LIN {X 0,Y 418.29,Z 497.008,A -85,B 0,C 180,E1 -10307.775,E2 -10307.775} C_VEL
LIN {X 0,Y 418.266,Z 497.012,A -85,B 0,C 180,E1 -10311.561,E2 -10311.561} C_VEL
LIN {X 0,Y 418.259,Z 497.011,A -85,B 0,C 180,E1 -10315.16,E2 -10315.16} C_VEL
LIN {X 0,Y 418.245,Z 497.014,A -85,B 0,C 180,E1 -10317.473,E2 -10317.473} C_VEL
LIN {X 0,Y 418.269,Z 497.007,A -85,B 0,C 180,E1 -10320.897,E2 -10320.897} C_VEL
LIN {X 0,Y 418.273,Z 497.008,A -85,B 0,C 180,E1 -10324.097,E2 -10324.097} C_VEL
LIN {X 0,Y 418.241,Z 497.014,A -85,B 0,C 180,E1 -10327.265,E2 -10327.265} C_VEL
LIN {X 0,Y 418.286,Z 497.005,A -85,B 0,C 180,E1 -10330.365,E2 -10330.365} C_VEL
LIN {X 0,Y 418.321,Z 497.004,A -85,B 0,C 180,E1 -10333.406,E2 -10333.406} C_VEL
LIN {X 0,Y 418.35,Z 496.998,A -85,B 0,C 180,E1 -10337,E2 -10337} C_VEL
LIN {X 0,Y 418.343,Z 496.998,A -85,B 0,C 180,E1 -10340.329,E2 -10340.329} C_VEL
LIN {X 0,Y 418.484,Z 496.982,A -85,B 0,C 180,E1 -10343.249,E2 -10343.249} C_VEL
LIN {X 0,Y 418.346,Z 496.999,A -85,B 0,C 180,E1 -10345.182,E2 -10345.182} C_VEL
LIN {X 0,Y 418.551,Z 496.974,A -85,B 0,C 180,E1 -10348.076,E2 -10348.076} C_VEL
LIN {X 0,Y 418.676,Z 496.959,A -85,B 0,C 180,E1 -10350,E2 -10350} C_VEL
LIN {X 0,Y 418.488,Z 496.984,A -85,B 0,C 180,E1 -10351.925,E2 -10351.925} C_VEL
LIN {X 0,Y 417.982,Z 497.048,A -85,B 0,C 180,E1 -10355.79,E2 -10355.79} C_VEL
LIN {X 0,Y 417.84,Z 497.118,A -85,B 0,C 180,E1 -10357.078,E2 -10357.078} C_VEL
LIN {X 0,Y 417.635,Z 500.157,A -85,B 0,C 180,E1 -10360.668,E2 -10360.668} C_VEL
LIN {X 0,Y 417.571,Z 502.391,A -85,B 0,C 180,E1 -10363.273,E2 -10363.273} C_VEL
LIN {X 0,Y 416.857,Z 502.803,A -85,B 0,C 180,E1 -10363.658,E2 -10363.658} C_VEL
LIN {X 0,Y 411.137,Z 504.383,A -85,B 0,C 180,E1 -10364.787,E2 -10364.787} C_VEL
LIN {X 0,Y 410.464,Z 504.792,A -85,B 0,C 180,E1 -10365.181,E2 -10365.181} C_VEL
LIN {X 0,Y 410.481,Z 505.038,A -85,B 0,C 180,E1 -10365.231,E2 -10365.231} C_VEL
LIN {X 0,Y 415.933,Z 520.618,A -85,B 0,C 180,E1 -10366,E2 -10366} C_VEL
LIN {X 0,Y 420.083,Z 534.2,A -85,B 0,C 180,E1 -10366.799,E2 -10366.799} C_VEL
LIN {X 0,Y 420.651,Z 537.197,A -85,B 0,C 180,E1 -10366.982,E2 -10366.982} C_VEL
LIN {X 0,Y 419.692,Z 552.291,A -85,B 0,C 180,E1 -10367.795,E2 -10367.795} C_VEL
LIN {X 0,Y 418.574,Z 565.955,A -85,B 0,C 180,E1 -10368.731,E2 -10368.731} C_VEL
LIN {X 0,Y 417.384,Z 578.751,A -85,B 0,C 180,E1 -10369.808,E2 -10369.808} C_VEL
LIN {X 0,Y 416.168,Z 591.539,A -85,B 0,C 180,E1 -10371.123,E2 -10371.123} C_VEL
LIN {X 0,Y 414.855,Z 603.015,A -85,B 0,C 180,E1 -10372.538,E2 -10372.538} C_VEL
LIN {X 0,Y 413.778,Z 613.302,A -85,B 0,C 180,E1 -10374.057,E2 -10374.057} C_VEL
LIN {X 0,Y 412.843,Z 621.821,A -85,B 0,C 180,E1 -10375.544,E2 -10375.544} C_VEL
LIN {X 0,Y 411.877,Z 630.973,A -85,B 0,C 180,E1 -10377.464,E2 -10377.464} C_VEL
LIN {X 0,Y 411.217,Z 638.263,A -85,B 0,C 180,E1 -10379.351,E2 -10379.351} C_VEL
LIN {X 0,Y 410.699,Z 643.934,A -85,B 0,C 180,E1 -10381.171,E2 -10381.171} C_VEL
LIN {X 0,Y 410.352,Z 648.94,A -85,B 0,C 180,E1 -10383.234,E2 -10383.234} C_VEL
LIN {X 0,Y 410.153,Z 651.623,A -85,B 0,C 180,E1 -10384.665,E2 -10384.665} C_VEL
LIN {X 0,Y 409.926,Z 654.472,A -85,B 0,C 180,E1 -10386.874,E2 -10386.874} C_VEL
LIN {X 0,Y 409.853,Z 655.422,A -85,B 0,C 180,E1 -10388.12,E2 -10388.12} C_VEL
LIN {X 0,Y 409.822,Z 655.948,A -85,B 0,C 180,E1 -10389.492,E2 -10389.492} C_VEL
LIN {X 0,Y 409.818,Z 655.929,A -85,B 0,C 180,E1 -10391.012,E2 -10391.012} C_VEL
LIN {X 0,Y 409.94,Z 654.61,A -85,B 0,C 180,E1 -10393.295,E2 -10393.295} C_VEL
LIN {X 0,Y 410.191,Z 652.038,A -85,B 0,C 180,E1 -10395.374,E2 -10395.374} C_VEL
LIN {X 0,Y 410.483,Z 648.227,A -85,B 0,C 180,E1 -10397.41,E2 -10397.41} C_VEL
LIN {X 0,Y 410.871,Z 643.027,A -85,B 0,C 180,E1 -10399.458,E2 -10399.458} C_VEL
LIN {X 0,Y 411.466,Z 636.994,A -85,B 0,C 180,E1 -10401.311,E2 -10401.311} C_VEL
LIN {X 0,Y 412.263,Z 629.191,A -85,B 0,C 180,E1 -10403.247,E2 -10403.247} C_VEL
LIN {X 0,Y 413.262,Z 620.342,A -85,B 0,C 180,E1 -10405.038,E2 -10405.038} C_VEL
LIN {X 0,Y 414.431,Z 610.328,A -85,B 0,C 180,E1 -10406.715,E2 -10406.715} C_VEL
LIN {X 0,Y 415.711,Z 599.27,A -85,B 0,C 180,E1 -10408.253,E2 -10408.253} C_VEL
LIN {X 0,Y 416.999,Z 587.412,A -85,B 0,C 180,E1 -10409.627,E2 -10409.627} C_VEL
LIN {X 0,Y 418.3,Z 574.278,A -85,B 0,C 180,E1 -10410.887,E2 -10410.887} C_VEL
LIN {X 0,Y 419.54,Z 560.488,A -85,B 0,C 180,E1 -10411.959,E2 -10411.959} C_VEL
LIN {X 0,Y 420.653,Z 546.6,A -85,B 0,C 180,E1 -10412.816,E2 -10412.816} C_VEL
LIN {X 0,Y 421.231,Z 537.263,A -85,B 0,C 180,E1 -10413.29,E2 -10413.29} C_VEL
LIN {X 0,Y 416.905,Z 523.396,A -85,B 0,C 180,E1 -10414.172,E2 -10414.172} C_VEL
LIN {X 0,Y 411.456,Z 509.384,A -85,B 0,C 180,E1 -10414.974,E2 -10414.974} C_VEL
LIN {X 0,Y 410.649,Z 506.752,A -85,B 0,C 180,E1 -10415.101,E2 -10415.101} C_VEL
LIN {X 0,Y 410.744,Z 504.603,A -85,B 0,C 180,E1 -10417.887,E2 -10417.887} C_VEL
LIN {X 0,Y 410.827,Z 502.253,A -85,B 0,C 180,E1 -10421.032,E2 -10421.032} C_VEL
LIN {X 0,Y 410.975,Z 499.978,A -85,B 0,C 180,E1 -10424.12,E2 -10424.12} C_VEL
LIN {X 0,Y 411.131,Z 497.904,A -85,B 0,C 180,E1 -10427.16,E2 -10427.16} C_VEL
LIN {X 0,Y 411.281,Z 497.883,A -85,B 0,C 180,E1 -10430.161,E2 -10430.161} C_VEL
LIN {X 0,Y 411.454,Z 497.857,A -85,B 0,C 180,E1 -10433.133,E2 -10433.133} C_VEL
LIN {X 0,Y 411.311,Z 497.876,A -85,B 0,C 180,E1 -10435.099,E2 -10435.099} C_VEL
LIN {X 0,Y 411.511,Z 497.851,A -85,B 0,C 180,E1 -10438.042,E2 -10438.042} C_VEL
LIN {X 0,Y 411.638,Z 497.835,A -85,B 0,C 180,E1 -10440,E2 -10440} C_VEL
LIN {X 0,Y 411.463,Z 497.858,A -85,B 0,C 180,E1 -10442.937,E2 -10442.937} C_VEL
LIN {X 0,Y 411.458,Z 497.859,A -85,B 0,C 180,E1 -10446.867,E2 -10446.867} C_VEL
LIN {X 0,Y 411.29,Z 497.877,A -85,B 0,C 180,E1 -10449.838,E2 -10449.838} C_VEL
LIN {X 0,Y 411.302,Z 497.876,A -85,B 0,C 180,E1 -10453.104,E2 -10453.104} C_VEL
LIN {X 0,Y 411.254,Z 497.882,A -85,B 0,C 180,E1 -10456.889,E2 -10456.889} C_VEL
LIN {X 0,Y 411.227,Z 497.884,A -85,B 0,C 180,E1 -10459.987,E2 -10459.987} C_VEL
LIN {X 0,Y 411.2,Z 497.887,A -85,B 0,C 180,E1 -10463.147,E2 -10463.147} C_VEL
LIN {X 0,Y 411.235,Z 497.885,A -85,B 0,C 180,E1 -10466.381,E2 -10466.381} C_VEL
LIN {X 0,Y 411.208,Z 497.891,A -85,B 0,C 180,E1 -10469.712,E2 -10469.712} C_VEL
LIN {X 0,Y 411.203,Z 497.889,A -85,B 0,C 180,E1 -10473.156,E2 -10473.156} C_VEL
LIN {X 0,Y 411.193,Z 497.892,A -85,B 0,C 180,E1 -10476.553,E2 -10476.553} C_VEL
LIN {X 0,Y 411.248,Z 498.032,A -85,B 0,C 180,E1 -10478.505,E2 -10478.505} C_VEL
LIN {X 0,Y 411.843,Z 501.621,A -85,B 0,C 180,E1 -10481.337,E2 -10481.337} C_VEL
LIN {X 0,Y 412.589,Z 505.831,A -85,B 0,C 180,E1 -10484.323,E2 -10484.323} C_VEL
LIN {X 0,Y 413.331,Z 510.237,A -85,B 0,C 180,E1 -10487.146,E2 -10487.146} C_VEL
LIN {X 0,Y 413.307,Z 513.645,A -85,B 0,C 180,E1 -10489.106,E2 -10489.106} C_VEL
LIN {X 0,Y 412.761,Z 519.39,A -85,B 0,C 180,E1 -10492.196,E2 -10492.196} C_VEL
LIN {X 0,Y 412.409,Z 524.702,A -85,B 0,C 180,E1 -10494.883,E2 -10494.883} C_VEL
LIN {X 0,Y 411.873,Z 532.35,A -85,B 0,C 180,E1 -10498.558,E2 -10498.558} C_VEL
LIN {X 0,Y 411.33,Z 539.833,A -85,B 0,C 180,E1 -10501.974,E2 -10501.974} C_VEL
LIN {X 0,Y 411.01,Z 546.461,A -85,B 0,C 180,E1 -10504.896,E2 -10504.896} C_VEL
LIN {X 0,Y 415.846,Z 565.472,A -85,B 0,C 180,E1 -10505.733,E2 -10505.733} C_VEL
LIN {X 0,Y 418.491,Z 580.052,A -85,B 0,C 180,E1 -10506.49,E2 -10506.49} C_VEL
LIN {X 0,Y 419.824,Z 589.116,A -85,B 0,C 180,E1 -10507.031,E2 -10507.031} C_VEL
LIN {X 0,Y 418.737,Z 602.749,A -85,B 0,C 180,E1 -10507.817,E2 -10507.817} C_VEL
LIN {X 0,Y 417.438,Z 616.129,A -85,B 0,C 180,E1 -10508.778,E2 -10508.778} C_VEL
LIN {X 0,Y 416.019,Z 629.933,A -85,B 0,C 180,E1 -10509.995,E2 -10509.995} C_VEL
LIN {X 0,Y 414.819,Z 641.407,A -85,B 0,C 180,E1 -10511.222,E2 -10511.222} C_VEL
LIN {X 0,Y 413.666,Z 653.061,A -85,B 0,C 180,E1 -10512.703,E2 -10512.703} C_VEL
LIN {X 0,Y 412.578,Z 662.893,A -85,B 0,C 180,E1 -10514.184,E2 -10514.184} C_VEL
LIN {X 0,Y 411.665,Z 672.58,A -85,B 0,C 180,E1 -10515.92,E2 -10515.92} C_VEL
LIN {X 0,Y 411.043,Z 680.676,A -85,B 0,C 180,E1 -10517.659,E2 -10517.659} C_VEL
LIN {X 0,Y 410.483,Z 688.249,A -85,B 0,C 180,E1 -10519.643,E2 -10519.643} C_VEL
LIN {X 0,Y 410.212,Z 694.284,A -85,B 0,C 180,E1 -10521.626,E2 -10521.626} C_VEL
LIN {X 0,Y 410.041,Z 699.25,A -85,B 0,C 180,E1 -10523.775,E2 -10523.775} C_VEL
LIN {X 0,Y 410.021,Z 701.523,A -85,B 0,C 180,E1 -10525.083,E2 -10525.083} C_VEL
LIN {X 0,Y 410.028,Z 703.932,A -85,B 0,C 180,E1 -10527.052,E2 -10527.052} C_VEL
LIN {X 0,Y 410.033,Z 705.156,A -85,B 0,C 180,E1 -10529.017,E2 -10529.017} C_VEL
LIN {X 0,Y 410.032,Z 705.191,A -85,B 0,C 180,E1 -10530.982,E2 -10530.982} C_VEL
LIN {X 0,Y 410.024,Z 704.011,A -85,B 0,C 180,E1 -10532.947,E2 -10532.947} C_VEL
LIN {X 0,Y 410.024,Z 701.648,A -85,B 0,C 180,E1 -10534.916,E2 -10534.916} C_VEL
LIN {X 0,Y 410.153,Z 698.06,A -85,B 0,C 180,E1 -10536.888,E2 -10536.888} C_VEL
LIN {X 0,Y 410.248,Z 693.142,A -85,B 0,C 180,E1 -10538.869,E2 -10538.869} C_VEL
LIN {X 0,Y 410.638,Z 686.783,A -85,B 0,C 180,E1 -10540.851,E2 -10540.851} C_VEL
LIN {X 0,Y 411.134,Z 678.795,A -85,B 0,C 180,E1 -10542.839,E2 -10542.839} C_VEL
LIN {X 0,Y 411.958,Z 670.307,A -85,B 0,C 180,E1 -10544.573,E2 -10544.573} C_VEL
LIN {X 0,Y 412.9,Z 660.081,A -85,B 0,C 180,E1 -10546.31,E2 -10546.31} C_VEL
LIN {X 0,Y 414.012,Z 649.665,A -85,B 0,C 180,E1 -10547.791,E2 -10547.791} C_VEL
LIN {X 0,Y 415.268,Z 637.192,A -85,B 0,C 180,E1 -10549.269,E2 -10549.269} C_VEL
LIN {X 0,Y 416.626,Z 624.734,A -85,B 0,C 180,E1 -10550.488,E2 -10550.488} C_VEL
LIN {X 0,Y 417.864,Z 611.122,A -85,B 0,C 180,E1 -10551.586,E2 -10551.586} C_VEL
LIN {X 0,Y 419.106,Z 597.196,A -85,B 0,C 180,E1 -10552.485,E2 -10552.485} C_VEL
LIN {X 0,Y 419.69,Z 588.951,A -85,B 0,C 180,E1 -10552.926,E2 -10552.926} C_VEL
LIN {X 0,Y 417.021,Z 573.601,A -85,B 0,C 180,E1 -10553.778,E2 -10553.778} C_VEL
LIN {X 0,Y 413.563,Z 558.078,A -85,B 0,C 180,E1 -10554.484,E2 -10554.484} C_VEL
LIN {X 0,Y 411.101,Z 548.197,A -85,B 0,C 180,E1 -10554.882,E2 -10554.882} C_VEL
LIN {X 0,Y 411.514,Z 541.099,A -85,B 0,C 180,E1 -10558.011,E2 -10558.011} C_VEL
LIN {X 0,Y 411.951,Z 533.541,A -85,B 0,C 180,E1 -10561.459,E2 -10561.459} C_VEL
LIN {X 0,Y 412.393,Z 527.674,A -85,B 0,C 180,E1 -10564.22,E2 -10564.22} C_VEL
LIN {X 0,Y 412.94,Z 520.375,A -85,B 0,C 180,E1 -10567.783,E2 -10567.783} C_VEL
LIN {X 0,Y 413.502,Z 514.296,A -85,B 0,C 180,E1 -10570.869,E2 -10570.869} C_VEL
LIN {X 0,Y 413.407,Z 510.324,A -85,B 0,C 180,E1 -10573.029,E2 -10573.029} C_VEL
LIN {X 0,Y 412.446,Z 504.612,A -85,B 0,C 180,E1 -10576.361,E2 -10576.361} C_VEL
LIN {X 0,Y 411.547,Z 499.514,A -85,B 0,C 180,E1 -10579.54,E2 -10579.54} C_VEL
LIN {X 0,Y 411.245,Z 497.886,A -85,B 0,C 180,E1 -10580.646,E2 -10580.646} C_VEL
LIN {X 0,Y 411.191,Z 497.891,A -85,B 0,C 180,E1 -10584.471,E2 -10584.471} C_VEL
LIN {X 0,Y 411.198,Z 497.89,A -85,B 0,C 180,E1 -10586.873,E2 -10586.873} C_VEL
LIN {X 0,Y 411.231,Z 497.883,A -85,B 0,C 180,E1 -10590.642,E2 -10590.642} C_VEL
LIN {X 0,Y 411.228,Z 497.888,A -85,B 0,C 180,E1 -10593.619,E2 -10593.619} C_VEL
LIN {X 0,Y 411.187,Z 497.89,A -85,B 0,C 180,E1 -10596.852,E2 -10596.852} C_VEL
LIN {X 0,Y 411.205,Z 497.888,A -85,B 0,C 180,E1 -10600.05,E2 -10600.05} C_VEL
LIN {X 0,Y 411.254,Z 497.883,A -85,B 0,C 180,E1 -10603.13,E2 -10603.13} C_VEL
LIN {X 0,Y 411.303,Z 497.875,A -85,B 0,C 180,E1 -10606.891,E2 -10606.891} C_VEL
LIN {X 0,Y 411.299,Z 497.876,A -85,B 0,C 180,E1 -10610.162,E2 -10610.162} C_VEL
LIN {X 0,Y 411.451,Z 497.859,A -85,B 0,C 180,E1 -10613.133,E2 -10613.133} C_VEL
LIN {X 0,Y 411.307,Z 497.876,A -85,B 0,C 180,E1 -10615.099,E2 -10615.099} C_VEL
LIN {X 0,Y 411.504,Z 497.851,A -85,B 0,C 180,E1 -10618.043,E2 -10618.043} C_VEL
LIN {X 0,Y 411.634,Z 497.835,A -85,B 0,C 180,E1 -10620,E2 -10620} C_VEL
LIN {X 0,Y 411.46,Z 497.856,A -85,B 0,C 180,E1 -10622.938,E2 -10622.938} C_VEL
LIN {X 0,Y 411.446,Z 497.856,A -85,B 0,C 180,E1 -10626.596,E2 -10626.596} C_VEL
LIN {X 0,Y 411.285,Z 497.88,A -85,B 0,C 180,E1 -10629.839,E2 -10629.839} C_VEL
LIN {X 0,Y 411.296,Z 497.878,A -85,B 0,C 180,E1 -10633.105,E2 -10633.105} C_VEL
LIN {X 0,Y 411.249,Z 497.881,A -85,B 0,C 180,E1 -10636.89,E2 -10636.89} C_VEL
LIN {X 0,Y 411.222,Z 497.887,A -85,B 0,C 180,E1 -10639.988,E2 -10639.988} C_VEL
LIN {X 0,Y 411.196,Z 497.891,A -85,B 0,C 180,E1 -10643.148,E2 -10643.148} C_VEL
LIN {X 0,Y 411.231,Z 497.883,A -85,B 0,C 180,E1 -10646.382,E2 -10646.382} C_VEL
LIN {X 0,Y 411.205,Z 497.891,A -85,B 0,C 180,E1 -10649.713,E2 -10649.713} C_VEL
LIN {X 0,Y 411.201,Z 497.89,A -85,B 0,C 180,E1 -10653.157,E2 -10653.157} C_VEL
LIN {X 0,Y 411.191,Z 497.888,A -85,B 0,C 180,E1 -10656.554,E2 -10656.554} C_VEL
LIN {X 0,Y 411.226,Z 497.889,A -85,B 0,C 180,E1 -10659.732,E2 -10659.732} C_VEL
LIN {X 0,Y 411.228,Z 497.886,A -85,B 0,C 180,E1 -10663.127,E2 -10663.127} C_VEL
LIN {X 0,Y 411.228,Z 497.887,A -85,B 0,C 180,E1 -10665.873,E2 -10665.873} C_VEL
LIN {X 0,Y 411.208,Z 497.886,A -85,B 0,C 180,E1 -10668.766,E2 -10668.766} C_VEL
LIN {X 0,Y 411.204,Z 497.889,A -85,B 0,C 180,E1 -10672.029,E2 -10672.029} C_VEL
LIN {X 0,Y 411.206,Z 497.891,A -85,B 0,C 180,E1 -10675.668,E2 -10675.668} C_VEL
LIN {X 0,Y 411.19,Z 497.891,A -85,B 0,C 180,E1 -10679.154,E2 -10679.154} C_VEL
LIN {X 0,Y 411.26,Z 497.88,A -85,B 0,C 180,E1 -10682.524,E2 -10682.524} C_VEL
LIN {X 0,Y 411.229,Z 497.888,A -85,B 0,C 180,E1 -10685.786,E2 -10685.786} C_VEL
LIN {X 0,Y 411.199,Z 497.888,A -85,B 0,C 180,E1 -10688.967,E2 -10688.967} C_VEL
LIN {X 0,Y 411.256,Z 497.882,A -85,B 0,C 180,E1 -10692.086,E2 -10692.086} C_VEL
LIN {X 0,Y 411.264,Z 497.881,A -85,B 0,C 180,E1 -10695.148,E2 -10695.148} C_VEL
LIN {X 0,Y 411.287,Z 497.878,A -85,B 0,C 180,E1 -10698.168,E2 -10698.168} C_VEL
LIN {X 0,Y 411.443,Z 497.858,A -85,B 0,C 180,E1 -10702.192,E2 -10702.192} C_VEL
LIN {X 0,Y 411.476,Z 497.855,A -85,B 0,C 180,E1 -10704.119,E2 -10704.119} C_VEL
LIN {X 0,Y 411.52,Z 497.85,A -85,B 0,C 180,E1 -10708.043,E2 -10708.043} C_VEL
LIN {X 0,Y 411.645,Z 497.835,A -85,B 0,C 180,E1 -10710,E2 -10710} C_VEL
LIN {X 0,Y 411.45,Z 497.86,A -85,B 0,C 180,E1 -10711.958,E2 -10711.958} C_VEL
LIN {X 0,Y 410.941,Z 497.924,A -85,B 0,C 180,E1 -10715.89,E2 -10715.89} C_VEL
LIN {X 0,Y 410.799,Z 497.969,A -85,B 0,C 180,E1 -10717.123,E2 -10717.123} C_VEL
LIN {X 0,Y 410.621,Z 500.232,A -85,B 0,C 180,E1 -10719.855,E2 -10719.855} C_VEL
LIN {X 0,Y 410.538,Z 502.812,A -85,B 0,C 180,E1 -10722.859,E2 -10722.859} C_VEL
LIN {X 0,Y 410.464,Z 504.792,A -85,B 0,C 180,E1 -10725.181,E2 -10725.181} C_VEL
LIN {X 0,Y 411.369,Z 505.402,A -85,B 0,C 180,E1 -10725.295,E2 -10725.295} C_VEL
LIN {X 0,Y 414.064,Z 508.494,A -85,B 0,C 180,E1 -10725.536,E2 -10725.536} C_VEL
LIN {X 0,Y 415.611,Z 511.968,A -85,B 0,C 180,E1 -10725.706,E2 -10725.706} C_VEL
LIN {X 0,Y 416.194,Z 517.03,A -85,B 0,C 180,E1 -10725.897,E2 -10725.897} C_VEL
LIN {X 0,Y 415.635,Z 521.611,A -85,B 0,C 180,E1 -10725.95,E2 -10725.95} C_VEL
LIN {X 0,Y 413.296,Z 529.526,A -85,B 0,C 180,E1 -10726.151,E2 -10726.151} C_VEL
LIN {X 0,Y 412.906,Z 532.831,A -85,B 0,C 180,E1 -10726.3,E2 -10726.3} C_VEL
LIN {X 0,Y 413.193,Z 534.941,A -85,B 0,C 180,E1 -10726.425,E2 -10726.425} C_VEL
LIN {X 0,Y 414.006,Z 538.808,A -85,B 0,C 180,E1 -10726.673,E2 -10726.673} C_VEL
LIN {X 0,Y 413.055,Z 553.102,A -85,B 0,C 180,E1 -10727.466,E2 -10727.466} C_VEL
LIN {X 0,Y 411.911,Z 566.481,A -85,B 0,C 180,E1 -10728.4,E2 -10728.4} C_VEL
LIN {X 0,Y 410.608,Z 579.831,A -85,B 0,C 180,E1 -10729.55,E2 -10729.55} C_VEL
LIN {X 0,Y 409.376,Z 592.351,A -85,B 0,C 180,E1 -10730.869,E2 -10730.869} C_VEL
LIN {X 0,Y 408.042,Z 603.489,A -85,B 0,C 180,E1 -10732.267,E2 -10732.267} C_VEL
LIN {X 0,Y 406.935,Z 613.382,A -85,B 0,C 180,E1 -10733.744,E2 -10733.744} C_VEL
LIN {X 0,Y 405.887,Z 622.569,A -85,B 0,C 180,E1 -10735.376,E2 -10735.376} C_VEL
LIN {X 0,Y 404.946,Z 631.301,A -85,B 0,C 180,E1 -10737.245,E2 -10737.245} C_VEL
LIN {X 0,Y 404.221,Z 638.5,A -85,B 0,C 180,E1 -10739.132,E2 -10739.132} C_VEL
LIN {X 0,Y 403.705,Z 643.887,A -85,B 0,C 180,E1 -10740.869,E2 -10740.869} C_VEL
LIN {X 0,Y 403.351,Z 648.436,A -85,B 0,C 180,E1 -10742.693,E2 -10742.693} C_VEL
LIN {X 0,Y 403.191,Z 650.843,A -85,B 0,C 180,E1 -10743.903,E2 -10743.903} C_VEL
LIN {X 0,Y 403.006,Z 652.842,A -85,B 0,C 180,E1 -10745.133,E2 -10745.133} C_VEL
LIN {X 0,Y 402.849,Z 654.698,A -85,B 0,C 180,E1 -10746.629,E2 -10746.629} C_VEL
LIN {X 0,Y 402.757,Z 656.254,A -85,B 0,C 180,E1 -10748.916,E2 -10748.916} C_VEL
LIN {X 0,Y 402.724,Z 656.466,A -85,B 0,C 180,E1 -10750.217,E2 -10750.217} C_VEL
LIN {X 0,Y 402.745,Z 656.187,A -85,B 0,C 180,E1 -10751.537,E2 -10751.537} C_VEL
LIN {X 0,Y 402.838,Z 655.408,A -85,B 0,C 180,E1 -10752.883,E2 -10752.883} C_VEL
LIN {X 0,Y 402.976,Z 653.999,A -85,B 0,C 180,E1 -10754.352,E2 -10754.352} C_VEL
LIN {X 0,Y 403.263,Z 650.841,A -85,B 0,C 180,E1 -10756.454,E2 -10756.454} C_VEL
LIN {X 0,Y 403.651,Z 646.288,A -85,B 0,C 180,E1 -10758.576,E2 -10758.576} C_VEL
LIN {X 0,Y 404.185,Z 640.494,A -85,B 0,C 180,E1 -10760.617,E2 -10760.617} C_VEL
LIN {X 0,Y 404.943,Z 633.389,A -85,B 0,C 180,E1 -10762.594,E2 -10762.594} C_VEL
LIN {X 0,Y 405.921,Z 625.107,A -85,B 0,C 180,E1 -10764.463,E2 -10764.463} C_VEL
LIN {X 0,Y 407.058,Z 615.553,A -85,B 0,C 180,E1 -10766.241,E2 -10766.241} C_VEL
LIN {X 0,Y 408.388,Z 604.754,A -85,B 0,C 180,E1 -10767.904,E2 -10767.904} C_VEL
LIN {X 0,Y 409.742,Z 593.312,A -85,B 0,C 180,E1 -10769.367,E2 -10769.367} C_VEL
LIN {X 0,Y 411.097,Z 580.984,A -85,B 0,C 180,E1 -10770.677,E2 -10770.677} C_VEL
LIN {X 0,Y 412.434,Z 567.966,A -85,B 0,C 180,E1 -10771.814,E2 -10771.814} C_VEL
LIN {X 0,Y 413.63,Z 554.227,A -85,B 0,C 180,E1 -10772.787,E2 -10772.787} C_VEL
LIN {X 0,Y 414.649,Z 539.89,A -85,B 0,C 180,E1 -10773.586,E2 -10773.586} C_VEL
LIN {X 0,Y 414.021,Z 536.459,A -85,B 0,C 180,E1 -10773.809,E2 -10773.809} C_VEL
LIN {X 0,Y 409.117,Z 521.383,A -85,B 0,C 180,E1 -10774.791,E2 -10774.791} C_VEL
LIN {X 0,Y 403.693,Z 507.937,A -85,B 0,C 180,E1 -10775.576,E2 -10775.576} C_VEL
LIN {X 0,Y 403.588,Z 507.237,A -85,B 0,C 180,E1 -10775.638,E2 -10775.638} C_VEL
LIN {X 0,Y 403.718,Z 505.038,A -85,B 0,C 180,E1 -10778.557,E2 -10778.557} C_VEL
LIN {X 0,Y 403.838,Z 502.696,A -85,B 0,C 180,E1 -10781.744,E2 -10781.744} C_VEL
LIN {X 0,Y 403.983,Z 500.441,A -85,B 0,C 180,E1 -10784.873,E2 -10784.873} C_VEL
LIN {X 0,Y 404.078,Z 499.029,A -85,B 0,C 180,E1 -10786.932,E2 -10786.932} C_VEL
LIN {X 0,Y 404.208,Z 498.764,A -85,B 0,C 180,E1 -10788.973,E2 -10788.973} C_VEL
LIN {X 0,Y 404.403,Z 498.738,A -85,B 0,C 180,E1 -10792.128,E2 -10792.128} C_VEL
LIN {X 0,Y 404.421,Z 498.736,A -85,B 0,C 180,E1 -10794.015,E2 -10794.015} C_VEL
LIN {X 0,Y 404.48,Z 498.727,A -85,B 0,C 180,E1 -10798.008,E2 -10798.008} C_VEL
LIN {X 0,Y 404.608,Z 498.711,A -85,B 0,C 180,E1 -10800,E2 -10800} C_VEL
LIN {X 0,Y 404.42,Z 498.735,A -85,B 0,C 180,E1 -10802.988,E2 -10802.988} C_VEL
LIN {X 0,Y 404.409,Z 498.736,A -85,B 0,C 180,E1 -10806.987,E2 -10806.987} C_VEL
LIN {X 0,Y 404.256,Z 498.753,A -85,B 0,C 180,E1 -10810.011,E2 -10810.011} C_VEL
LIN {X 0,Y 404.263,Z 498.752,A -85,B 0,C 180,E1 -10813.211,E2 -10813.211} C_VEL
LIN {X 0,Y 404.212,Z 498.758,A -85,B 0,C 180,E1 -10817.007,E2 -10817.007} C_VEL
LIN {X 0,Y 404.16,Z 498.768,A -85,B 0,C 180,E1 -10820.351,E2 -10820.351} C_VEL
LIN {X 0,Y 404.166,Z 498.763,A -85,B 0,C 180,E1 -10823.574,E2 -10823.574} C_VEL
LIN {X 0,Y 404.181,Z 498.764,A -85,B 0,C 180,E1 -10825.766,E2 -10825.766} C_VEL
LIN {X 0,Y 404.195,Z 498.764,A -85,B 0,C 180,E1 -10827.999,E2 -10827.999} C_VEL
LIN {X 0,Y 404.14,Z 498.77,A -85,B 0,C 180,E1 -10831.559,E2 -10831.559} C_VEL
LIN {X 0,Y 404.183,Z 498.764,A -85,B 0,C 180,E1 -10835.016,E2 -10835.016} C_VEL
LIN {X 0,Y 404.167,Z 498.875,A -85,B 0,C 180,E1 -10837.888,E2 -10837.888} C_VEL
LIN {X 0,Y 404.69,Z 501.567,A -85,B 0,C 180,E1 -10840.172,E2 -10840.172} C_VEL
LIN {X 0,Y 405.524,Z 506.611,A -85,B 0,C 180,E1 -10843.886,E2 -10843.886} C_VEL
LIN {X 0,Y 406.233,Z 510.723,A -85,B 0,C 180,E1 -10846.603,E2 -10846.603} C_VEL
LIN {X 0,Y 406.408,Z 513.041,A -85,B 0,C 180,E1 -10848.038,E2 -10848.038} C_VEL
LIN {X 0,Y 405.925,Z 518.639,A -85,B 0,C 180,E1 -10851.179,E2 -10851.179} C_VEL
LIN {X 0,Y 405.422,Z 525.101,A -85,B 0,C 180,E1 -10854.562,E2 -10854.562} C_VEL
LIN {X 0,Y 404.945,Z 530.94,A -85,B 0,C 180,E1 -10857.451,E2 -10857.451} C_VEL
LIN {X 0,Y 404.548,Z 536.955,A -85,B 0,C 180,E1 -10860.299,E2 -10860.299} C_VEL
LIN {X 0,Y 404.099,Z 544.343,A -85,B 0,C 180,E1 -10863.673,E2 -10863.673} C_VEL
LIN {X 0,Y 403.992,Z 545.989,A -85,B 0,C 180,E1 -10864.408,E2 -10864.408} C_VEL
LIN {X 0,Y 408.505,Z 563.256,A -85,B 0,C 180,E1 -10865.187,E2 -10865.187} C_VEL
LIN {X 0,Y 411.418,Z 577.948,A -85,B 0,C 180,E1 -10865.967,E2 -10865.967} C_VEL
LIN {X 0,Y 413.168,Z 590.212,A -85,B 0,C 180,E1 -10866.713,E2 -10866.713} C_VEL
LIN {X 0,Y 411.923,Z 604.633,A -85,B 0,C 180,E1 -10867.586,E2 -10867.586} C_VEL
LIN {X 0,Y 410.628,Z 617.372,A -85,B 0,C 180,E1 -10868.541,E2 -10868.541} C_VEL
LIN {X 0,Y 409.15,Z 630.825,A -85,B 0,C 180,E1 -10869.776,E2 -10869.776} C_VEL
LIN {X 0,Y 407.829,Z 642.875,A -85,B 0,C 180,E1 -10871.113,E2 -10871.113} C_VEL
LIN {X 0,Y 406.606,Z 654.458,A -85,B 0,C 180,E1 -10872.653,E2 -10872.653} C_VEL
LIN {X 0,Y 405.371,Z 665.473,A -85,B 0,C 180,E1 -10874.411,E2 -10874.411} C_VEL
LIN {X 0,Y 404.471,Z 674.794,A -85,B 0,C 180,E1 -10876.203,E2 -10876.203} C_VEL
LIN {X 0,Y 403.838,Z 682.334,A -85,B 0,C 180,E1 -10877.946,E2 -10877.946} C_VEL
LIN {X 0,Y 403.286,Z 689.494,A -85,B 0,C 180,E1 -10879.964,E2 -10879.964} C_VEL
LIN {X 0,Y 403.078,Z 695.147,A -85,B 0,C 180,E1 -10881.981,E2 -10881.981} C_VEL
LIN {X 0,Y 402.936,Z 699.433,A -85,B 0,C 180,E1 -10883.992,E2 -10883.992} C_VEL
LIN {X 0,Y 402.879,Z 702.449,A -85,B 0,C 180,E1 -10885.998,E2 -10885.998} C_VEL
LIN {X 0,Y 402.971,Z 704.265,A -85,B 0,C 180,E1 -10888.001,E2 -10888.001} C_VEL
LIN {X 0,Y 402.963,Z 704.904,A -85,B 0,C 180,E1 -10889.999,E2 -10889.999} C_VEL
LIN {X 0,Y 402.97,Z 704.32,A -85,B 0,C 180,E1 -10891.998,E2 -10891.998} C_VEL
LIN {X 0,Y 402.87,Z 702.543,A -85,B 0,C 180,E1 -10894.001,E2 -10894.001} C_VEL
LIN {X 0,Y 402.984,Z 699.573,A -85,B 0,C 180,E1 -10896.006,E2 -10896.006} C_VEL
LIN {X 0,Y 403.078,Z 695.324,A -85,B 0,C 180,E1 -10898.017,E2 -10898.017} C_VEL
LIN {X 0,Y 403.286,Z 689.692,A -85,B 0,C 180,E1 -10900.035,E2 -10900.035} C_VEL
LIN {X 0,Y 403.839,Z 682.539,A -85,B 0,C 180,E1 -10902.053,E2 -10902.053} C_VEL
LIN {X 0,Y 404.475,Z 675.009,A -85,B 0,C 180,E1 -10903.796,E2 -10903.796} C_VEL
LIN {X 0,Y 405.373,Z 665.673,A -85,B 0,C 180,E1 -10905.588,E2 -10905.588} C_VEL
LIN {X 0,Y 406.639,Z 654.56,A -85,B 0,C 180,E1 -10907.345,E2 -10907.345} C_VEL
LIN {X 0,Y 407.825,Z 642.842,A -85,B 0,C 180,E1 -10908.888,E2 -10908.888} C_VEL
LIN {X 0,Y 409.14,Z 630.638,A -85,B 0,C 180,E1 -10910.223,E2 -10910.223} C_VEL
LIN {X 0,Y 410.411,Z 618.372,A -85,B 0,C 180,E1 -10911.338,E2 -10911.338} C_VEL
LIN {X 0,Y 411.844,Z 603.969,A -85,B 0,C 180,E1 -10912.402,E2 -10912.402} C_VEL
LIN {X 0,Y 412.988,Z 589.857,A -85,B 0,C 180,E1 -10913.229,E2 -10913.229} C_VEL
LIN {X 0,Y 410.247,Z 573.892,A -85,B 0,C 180,E1 -10914.149,E2 -10914.149} C_VEL
LIN {X 0,Y 406.646,Z 557.983,A -85,B 0,C 180,E1 -10914.9,E2 -10914.9} C_VEL
LIN {X 0,Y 404.09,Z 547.804,A -85,B 0,C 180,E1 -10915.312,E2 -10915.312} C_VEL
LIN {X 0,Y 404.502,Z 540.697,A -85,B 0,C 180,E1 -10918.54,E2 -10918.54} C_VEL
LIN {X 0,Y 404.93,Z 533.843,A -85,B 0,C 180,E1 -10921.74,E2 -10921.74} C_VEL
LIN {X 0,Y 405.365,Z 528.511,A -85,B 0,C 180,E1 -10924.295,E2 -10924.295} C_VEL
LIN {X 0,Y 406.084,Z 520.002,A -85,B 0,C 180,E1 -10928.537,E2 -10928.537} C_VEL
LIN {X 0,Y 406.513,Z 515.155,A -85,B 0,C 180,E1 -10931.067,E2 -10931.067} C_VEL
LIN {X 0,Y 406.336,Z 510.917,A -85,B 0,C 180,E1 -10933.412,E2 -10933.412} C_VEL
LIN {X 0,Y 405.354,Z 505.371,A -85,B 0,C 180,E1 -10936.733,E2 -10936.733} C_VEL
LIN {X 0,Y 404.457,Z 500.266,A -85,B 0,C 180,E1 -10939.99,E2 -10939.99} C_VEL
LIN {X 0,Y 404.174,Z 498.767,A -85,B 0,C 180,E1 -10941.086,E2 -10941.086} C_VEL
LIN {X 0,Y 404.177,Z 498.764,A -85,B 0,C 180,E1 -10944.983,E2 -10944.983} C_VEL
LIN {X 0,Y 404.137,Z 498.767,A -85,B 0,C 180,E1 -10948.554,E2 -10948.554} C_VEL
LIN {X 0,Y 404.189,Z 498.762,A -85,B 0,C 180,E1 -10952,E2 -10952} C_VEL
LIN {X 0,Y 404.165,Z 498.768,A -85,B 0,C 180,E1 -10955.334,E2 -10955.334} C_VEL
LIN {X 0,Y 404.128,Z 498.768,A -85,B 0,C 180,E1 -10958.58,E2 -10958.58} C_VEL
LIN {X 0,Y 404.2,Z 498.763,A -85,B 0,C 180,E1 -10961.762,E2 -10961.762} C_VEL
LIN {X 0,Y 404.202,Z 498.759,A -85,B 0,C 180,E1 -10964.882,E2 -10964.882} C_VEL
LIN {X 0,Y 404.26,Z 498.754,A -85,B 0,C 180,E1 -10967.959,E2 -10967.959} C_VEL
LIN {X 0,Y 404.423,Z 498.732,A -85,B 0,C 180,E1 -10972.1,E2 -10972.1} C_VEL
LIN {X 0,Y 404.416,Z 498.733,A -85,B 0,C 180,E1 -10974.015,E2 -10974.015} C_VEL
LIN {X 0,Y 404.473,Z 498.727,A -85,B 0,C 180,E1 -10978.009,E2 -10978.009} C_VEL
LIN {X 0,Y 404.603,Z 498.711,A -85,B 0,C 180,E1 -10980,E2 -10980} C_VEL
LIN {X 0,Y 404.417,Z 498.733,A -85,B 0,C 180,E1 -10982.989,E2 -10982.989} C_VEL
LIN {X 0,Y 404.394,Z 498.734,A -85,B 0,C 180,E1 -10986.593,E2 -10986.593} C_VEL
LIN {X 0,Y 404.282,Z 498.75,A -85,B 0,C 180,E1 -10989.002,E2 -10989.002} C_VEL
LIN {X 0,Y 404.248,Z 498.755,A -85,B 0,C 180,E1 -10992.042,E2 -10992.042} C_VEL
LIN {X 0,Y 404.197,Z 498.762,A -85,B 0,C 180,E1 -10995.119,E2 -10995.119} C_VEL
LIN {X 0,Y 404.202,Z 498.759,A -85,B 0,C 180,E1 -10998.239,E2 -10998.239} C_VEL
LIN {X 0,Y 404.131,Z 498.772,A -85,B 0,C 180,E1 -11001.42,E2 -11001.42} C_VEL
LIN {X 0,Y 404.17,Z 498.763,A -85,B 0,C 180,E1 -11004.667,E2 -11004.667} C_VEL
LIN {X 0,Y 404.191,Z 498.762,A -85,B 0,C 180,E1 -11008.001,E2 -11008.001} C_VEL
LIN {X 0,Y 404.141,Z 498.772,A -85,B 0,C 180,E1 -11011.561,E2 -11011.561} C_VEL
LIN {X 0,Y 404.18,Z 498.763,A -85,B 0,C 180,E1 -11015.017,E2 -11015.017} C_VEL
LIN {X 0,Y 404.16,Z 498.764,A -85,B 0,C 180,E1 -11018.757,E2 -11018.757} C_VEL
LIN {X 0,Y 404.188,Z 498.765,A -85,B 0,C 180,E1 -11021.612,E2 -11021.612} C_VEL
LIN {X 0,Y 404.198,Z 498.759,A -85,B 0,C 180,E1 -11024.531,E2 -11024.531} C_VEL
LIN {X 0,Y 404.205,Z 498.762,A -85,B 0,C 180,E1 -11027.306,E2 -11027.306} C_VEL
LIN {X 0,Y 404.167,Z 498.766,A -85,B 0,C 180,E1 -11029.957,E2 -11029.957} C_VEL
LIN {X 0,Y 404.14,Z 498.769,A -85,B 0,C 180,E1 -11033.125,E2 -11033.125} C_VEL
LIN {X 0,Y 404.145,Z 498.767,A -85,B 0,C 180,E1 -11036.189,E2 -11036.189} C_VEL
LIN {X 0,Y 404.146,Z 498.771,A -85,B 0,C 180,E1 -11039.716,E2 -11039.716} C_VEL
LIN {X 0,Y 404.197,Z 498.761,A -85,B 0,C 180,E1 -11043.124,E2 -11043.124} C_VEL
LIN {X 0,Y 404.179,Z 498.765,A -85,B 0,C 180,E1 -11045.336,E2 -11045.336} C_VEL
LIN {X 0,Y 404.141,Z 498.766,A -85,B 0,C 180,E1 -11048.582,E2 -11048.582} C_VEL
LIN {X 0,Y 404.214,Z 498.762,A -85,B 0,C 180,E1 -11051.763,E2 -11051.763} C_VEL
LIN {X 0,Y 404.21,Z 498.758,A -85,B 0,C 180,E1 -11054.883,E2 -11054.883} C_VEL
LIN {X 0,Y 404.26,Z 498.755,A -85,B 0,C 180,E1 -11057.959,E2 -11057.959} C_VEL
LIN {X 0,Y 404.27,Z 498.751,A -85,B 0,C 180,E1 -11060.999,E2 -11060.999} C_VEL
LIN {X 0,Y 404.423,Z 498.734,A -85,B 0,C 180,E1 -11064.016,E2 -11064.016} C_VEL
LIN {X 0,Y 404.489,Z 498.726,A -85,B 0,C 180,E1 -11068.009,E2 -11068.009} C_VEL
LIN {X 0,Y 404.614,Z 498.71,A -85,B 0,C 180,E1 -11070.001,E2 -11070.001} C_VEL
LIN {X 0,Y 404.412,Z 498.736,A -85,B 0,C 180,E1 -11071.992,E2 -11071.992} C_VEL
LIN {X 0,Y 403.901,Z 498.801,A -85,B 0,C 180,E1 -11075.993,E2 -11075.993} C_VEL
LIN {X 0,Y 403.761,Z 498.823,A -85,B 0,C 180,E1 -11077.174,E2 -11077.174} C_VEL
LIN {X 0,Y 403.556,Z 501.208,A -85,B 0,C 180,E1 -11080.03,E2 -11080.03} C_VEL
LIN {X 0,Y 403.461,Z 503.783,A -85,B 0,C 180,E1 -11083.088,E2 -11083.088} C_VEL
LIN {X 0,Y 403.406,Z 505.213,A -85,B 0,C 180,E1 -11084.761,E2 -11084.761} C_VEL
LIN {X 0,Y 405.428,Z 511.037,A -85,B 0,C 180,E1 -11085.056,E2 -11085.056} C_VEL
LIN {X 0,Y 410.426,Z 525.605,A -85,B 0,C 180,E1 -11085.849,E2 -11085.849} C_VEL
LIN {X 0,Y 413.193,Z 534.941,A -85,B 0,C 180,E1 -11086.425,E2 -11086.425} C_VEL
LIN {X 0,Y 413.294,Z 537.952,A -85,B 0,C 180,E1 -11086.583,E2 -11086.583} C_VEL
LIN {X 0,Y 411.822,Z 542.242,A -85,B 0,C 180,E1 -11086.72,E2 -11086.72} C_VEL
LIN {X 0,Y 407.314,Z 550.681,A -85,B 0,C 180,E1 -11086.959,E2 -11086.959} C_VEL
LIN {X 0,Y 406.419,Z 554.435,A -85,B 0,C 180,E1 -11087.161,E2 -11087.161} C_VEL
LIN {X 0,Y 405.3,Z 566.721,A -85,B 0,C 180,E1 -11088.036,E2 -11088.036} C_VEL
LIN {X 0,Y 403.993,Z 579.74,A -85,B 0,C 180,E1 -11089.169,E2 -11089.169} C_VEL
LIN {X 0,Y 402.76,Z 591.653,A -85,B 0,C 180,E1 -11090.426,E2 -11090.426} C_VEL
LIN {X 0,Y 401.241,Z 603.807,A -85,B 0,C 180,E1 -11091.964,E2 -11091.964} C_VEL
LIN {X 0,Y 400.027,Z 614.253,A -85,B 0,C 180,E1 -11093.559,E2 -11093.559} C_VEL
LIN {X 0,Y 398.914,Z 623.458,A -85,B 0,C 180,E1 -11095.232,E2 -11095.232} C_VEL
LIN {X 0,Y 397.973,Z 631.754,A -85,B 0,C 180,E1 -11097.048,E2 -11097.048} C_VEL
LIN {X 0,Y 397.171,Z 639.466,A -85,B 0,C 180,E1 -11099.118,E2 -11099.118} C_VEL
LIN {X 0,Y 396.643,Z 644.846,A -85,B 0,C 180,E1 -11100.92,E2 -11100.92} C_VEL
LIN {X 0,Y 396.293,Z 649.193,A -85,B 0,C 180,E1 -11102.745,E2 -11102.745} C_VEL
LIN {X 0,Y 395.992,Z 652.609,A -85,B 0,C 180,E1 -11104.606,E2 -11104.606} C_VEL
LIN {X 0,Y 395.737,Z 655.445,A -85,B 0,C 180,E1 -11106.949,E2 -11106.949} C_VEL
LIN {X 0,Y 395.669,Z 656.526,A -85,B 0,C 180,E1 -11108.597,E2 -11108.597} C_VEL
LIN {X 0,Y 395.664,Z 656.897,A -85,B 0,C 180,E1 -11110.2,E2 -11110.2} C_VEL
LIN {X 0,Y 395.714,Z 656.217,A -85,B 0,C 180,E1 -11112.445,E2 -11112.445} C_VEL
LIN {X 0,Y 395.936,Z 654.052,A -85,B 0,C 180,E1 -11114.763,E2 -11114.763} C_VEL
LIN {X 0,Y 396.226,Z 651.158,A -85,B 0,C 180,E1 -11116.654,E2 -11116.654} C_VEL
LIN {X 0,Y 396.598,Z 647.111,A -85,B 0,C 180,E1 -11118.579,E2 -11118.579} C_VEL
LIN {X 0,Y 397.069,Z 642.167,A -85,B 0,C 180,E1 -11120.417,E2 -11120.417} C_VEL
LIN {X 0,Y 397.779,Z 636.056,A -85,B 0,C 180,E1 -11122.253,E2 -11122.253} C_VEL
LIN {X 0,Y 398.709,Z 628.186,A -85,B 0,C 180,E1 -11124.177,E2 -11124.177} C_VEL
LIN {X 0,Y 399.929,Z 618.612,A -85,B 0,C 180,E1 -11126.085,E2 -11126.085} C_VEL
LIN {X 0,Y 401.322,Z 607.996,A -85,B 0,C 180,E1 -11127.826,E2 -11127.826} C_VEL
LIN {X 0,Y 402.608,Z 597.656,A -85,B 0,C 180,E1 -11129.249,E2 -11129.249} C_VEL
LIN {X 0,Y 404.008,Z 586.014,A -85,B 0,C 180,E1 -11130.587,E2 -11130.587} C_VEL
LIN {X 0,Y 405.538,Z 572.164,A -85,B 0,C 180,E1 -11131.897,E2 -11131.897} C_VEL
LIN {X 0,Y 406.861,Z 558.154,A -85,B 0,C 180,E1 -11132.966,E2 -11132.966} C_VEL
LIN {X 0,Y 407.989,Z 544.296,A -85,B 0,C 180,E1 -11133.804,E2 -11133.804} C_VEL
LIN {X 0,Y 408.166,Z 541.316,A -85,B 0,C 180,E1 -11133.954,E2 -11133.954} C_VEL
LIN {X 0,Y 406.077,Z 533.341,A -85,B 0,C 180,E1 -11134.511,E2 -11134.511} C_VEL
LIN {X 0,Y 401.6,Z 520.387,A -85,B 0,C 180,E1 -11135.372,E2 -11135.372} C_VEL
LIN {X 0,Y 396.715,Z 508.613,A -85,B 0,C 180,E1 -11136.093,E2 -11136.093} C_VEL
LIN {X 0,Y 396.571,Z 507.764,A -85,B 0,C 180,E1 -11136.153,E2 -11136.153} C_VEL
LIN {X 0,Y 396.727,Z 505.023,A -85,B 0,C 180,E1 -11139.865,E2 -11139.865} C_VEL
LIN {X 0,Y 396.893,Z 502.403,A -85,B 0,C 180,E1 -11143.541,E2 -11143.541} C_VEL
LIN {X 0,Y 397.067,Z 500.169,A -85,B 0,C 180,E1 -11146.775,E2 -11146.775} C_VEL
LIN {X 0,Y 397.068,Z 499.656,A -85,B 0,C 180,E1 -11147.737,E2 -11147.737} C_VEL
LIN {X 0,Y 397.247,Z 499.628,A -85,B 0,C 180,E1 -11150.838,E2 -11150.838} C_VEL
LIN {X 0,Y 397.372,Z 499.614,A -85,B 0,C 180,E1 -11153.908,E2 -11153.908} C_VEL
LIN {X 0,Y 397.449,Z 499.603,A -85,B 0,C 180,E1 -11157.973,E2 -11157.973} C_VEL
LIN {X 0,Y 397.577,Z 499.587,A -85,B 0,C 180,E1 -11160,E2 -11160} C_VEL
LIN {X 0,Y 397.378,Z 499.612,A -85,B 0,C 180,E1 -11163.041,E2 -11163.041} C_VEL
LIN {X 0,Y 397.361,Z 499.613,A -85,B 0,C 180,E1 -11167.111,E2 -11167.111} C_VEL
LIN {X 0,Y 397.215,Z 499.63,A -85,B 0,C 180,E1 -11170.191,E2 -11170.191} C_VEL
LIN {X 0,Y 397.223,Z 499.628,A -85,B 0,C 180,E1 -11173.321,E2 -11173.321} C_VEL
LIN {X 0,Y 397.179,Z 499.634,A -85,B 0,C 180,E1 -11177.155,E2 -11177.155} C_VEL
LIN {X 0,Y 397.099,Z 499.646,A -85,B 0,C 180,E1 -11180.73,E2 -11180.73} C_VEL
LIN {X 0,Y 397.13,Z 499.643,A -85,B 0,C 180,E1 -11184.018,E2 -11184.018} C_VEL
LIN {X 0,Y 397.192,Z 499.634,A -85,B 0,C 180,E1 -11187.39,E2 -11187.39} C_VEL
LIN {X 0,Y 397.082,Z 499.65,A -85,B 0,C 180,E1 -11190.882,E2 -11190.882} C_VEL
LIN {X 0,Y 397.123,Z 499.643,A -85,B 0,C 180,E1 -11194.493,E2 -11194.493} C_VEL
LIN {X 0,Y 397.118,Z 499.673,A -85,B 0,C 180,E1 -11197.214,E2 -11197.214} C_VEL
LIN {X 0,Y 397.829,Z 503.577,A -85,B 0,C 180,E1 -11200.569,E2 -11200.569} C_VEL
LIN {X 0,Y 398.521,Z 507.746,A -85,B 0,C 180,E1 -11203.694,E2 -11203.694} C_VEL
LIN {X 0,Y 399.277,Z 512.106,A -85,B 0,C 180,E1 -11206.649,E2 -11206.649} C_VEL
LIN {X 0,Y 399.423,Z 514.351,A -85,B 0,C 180,E1 -11208.039,E2 -11208.039} C_VEL
LIN {X 0,Y 398.968,Z 519.18,A -85,B 0,C 180,E1 -11210.812,E2 -11210.812} C_VEL
LIN {X 0,Y 398.425,Z 525.869,A -85,B 0,C 180,E1 -11214.402,E2 -11214.402} C_VEL
LIN {X 0,Y 397.908,Z 531.808,A -85,B 0,C 180,E1 -11217.405,E2 -11217.405} C_VEL
LIN {X 0,Y 397.492,Z 537.831,A -85,B 0,C 180,E1 -11220.326,E2 -11220.326} C_VEL
LIN {X 0,Y 397.02,Z 545.439,A -85,B 0,C 180,E1 -11223.87,E2 -11223.87} C_VEL
LIN {X 0,Y 402.092,Z 564.819,A -85,B 0,C 180,E1 -11224.804,E2 -11224.804} C_VEL
LIN {X 0,Y 404.96,Z 579.748,A -85,B 0,C 180,E1 -11225.641,E2 -11225.641} C_VEL
LIN {X 0,Y 406.522,Z 591.325,A -85,B 0,C 180,E1 -11226.386,E2 -11226.386} C_VEL
LIN {X 0,Y 405.146,Z 606.244,A -85,B 0,C 180,E1 -11227.331,E2 -11227.331} C_VEL
LIN {X 0,Y 403.684,Z 619.951,A -85,B 0,C 180,E1 -11228.421,E2 -11228.421} C_VEL
LIN {X 0,Y 402.186,Z 632.879,A -85,B 0,C 180,E1 -11229.677,E2 -11229.677} C_VEL
LIN {X 0,Y 400.809,Z 644.706,A -85,B 0,C 180,E1 -11231.061,E2 -11231.061} C_VEL
LIN {X 0,Y 399.546,Z 655.746,A -85,B 0,C 180,E1 -11232.6,E2 -11232.6} C_VEL
LIN {X 0,Y 398.454,Z 665.074,A -85,B 0,C 180,E1 -11234.134,E2 -11234.134} C_VEL
LIN {X 0,Y 397.498,Z 674.265,A -85,B 0,C 180,E1 -11235.93,E2 -11235.93} C_VEL
LIN {X 0,Y 396.832,Z 681.924,A -85,B 0,C 180,E1 -11237.729,E2 -11237.729} C_VEL
LIN {X 0,Y 396.23,Z 689.081,A -85,B 0,C 180,E1 -11239.783,E2 -11239.783} C_VEL
LIN {X 0,Y 396.011,Z 694.733,A -85,B 0,C 180,E1 -11241.837,E2 -11241.837} C_VEL
LIN {X 0,Y 395.859,Z 699.015,A -85,B 0,C 180,E1 -11243.885,E2 -11243.885} C_VEL
LIN {X 0,Y 395.798,Z 702.028,A -85,B 0,C 180,E1 -11245.927,E2 -11245.927} C_VEL
LIN {X 0,Y 395.9,Z 703.841,A -85,B 0,C 180,E1 -11247.965,E2 -11247.965} C_VEL
LIN {X 0,Y 395.884,Z 704.476,A -85,B 0,C 180,E1 -11249.999,E2 -11249.999} C_VEL
LIN {X 0,Y 395.899,Z 703.891,A -85,B 0,C 180,E1 -11252.034,E2 -11252.034} C_VEL
LIN {X 0,Y 395.791,Z 702.106,A -85,B 0,C 180,E1 -11254.072,E2 -11254.072} C_VEL
LIN {X 0,Y 395.929,Z 698.863,A -85,B 0,C 180,E1 -11256.263,E2 -11256.263} C_VEL
LIN {X 0,Y 396.012,Z 694.866,A -85,B 0,C 180,E1 -11258.161,E2 -11258.161} C_VEL
LIN {X 0,Y 396.23,Z 689.217,A -85,B 0,C 180,E1 -11260.216,E2 -11260.216} C_VEL
LIN {X 0,Y 396.829,Z 682.045,A -85,B 0,C 180,E1 -11262.27,E2 -11262.27} C_VEL
LIN {X 0,Y 397.499,Z 674.372,A -85,B 0,C 180,E1 -11264.069,E2 -11264.069} C_VEL
LIN {X 0,Y 398.434,Z 665.142,A -85,B 0,C 180,E1 -11265.866,E2 -11265.866} C_VEL
LIN {X 0,Y 399.576,Z 655.728,A -85,B 0,C 180,E1 -11267.397,E2 -11267.397} C_VEL
LIN {X 0,Y 400.81,Z 644.504,A -85,B 0,C 180,E1 -11268.941,E2 -11268.941} C_VEL
LIN {X 0,Y 402.14,Z 632.459,A -85,B 0,C 180,E1 -11270.324,E2 -11270.324} C_VEL
LIN {X 0,Y 403.579,Z 619.171,A -85,B 0,C 180,E1 -11271.584,E2 -11271.584} C_VEL
LIN {X 0,Y 405.039,Z 605.177,A -85,B 0,C 180,E1 -11272.656,E2 -11272.656} C_VEL
LIN {X 0,Y 406.264,Z 590.862,A -85,B 0,C 180,E1 -11273.531,E2 -11273.531} C_VEL
LIN {X 0,Y 403.649,Z 575.364,A -85,B 0,C 180,E1 -11274.465,E2 -11274.465} C_VEL
LIN {X 0,Y 400.263,Z 560.095,A -85,B 0,C 180,E1 -11275.226,E2 -11275.226} C_VEL
LIN {X 0,Y 397.088,Z 547.442,A -85,B 0,C 180,E1 -11275.766,E2 -11275.766} C_VEL
LIN {X 0,Y 397.486,Z 540.259,A -85,B 0,C 180,E1 -11279.092,E2 -11279.092} C_VEL
LIN {X 0,Y 397.922,Z 534.093,A -85,B 0,C 180,E1 -11282.031,E2 -11282.031} C_VEL
LIN {X 0,Y 398.331,Z 529.33,A -85,B 0,C 180,E1 -11284.373,E2 -11284.373} C_VEL
LIN {X 0,Y 398.957,Z 522.036,A -85,B 0,C 180,E1 -11288.064,E2 -11288.064} C_VEL
LIN {X 0,Y 399.538,Z 515.872,A -85,B 0,C 180,E1 -11291.336,E2 -11291.336} C_VEL
LIN {X 0,Y 399.377,Z 512.335,A -85,B 0,C 180,E1 -11293.336,E2 -11293.336} C_VEL
LIN {X 0,Y 398.461,Z 507.057,A -85,B 0,C 180,E1 -11296.538,E2 -11296.538} C_VEL
LIN {X 0,Y 397.642,Z 502.503,A -85,B 0,C 180,E1 -11299.461,E2 -11299.461} C_VEL
LIN {X 0,Y 397.131,Z 499.643,A -85,B 0,C 180,E1 -11301.425,E2 -11301.425} C_VEL
LIN {X 0,Y 397.112,Z 499.644,A -85,B 0,C 180,E1 -11304.496,E2 -11304.496} C_VEL
LIN {X 0,Y 397.072,Z 499.649,A -85,B 0,C 180,E1 -11307.928,E2 -11307.928} C_VEL
LIN {X 0,Y 397.118,Z 499.646,A -85,B 0,C 180,E1 -11311.456,E2 -11311.456} C_VEL
LIN {X 0,Y 397.143,Z 499.638,A -85,B 0,C 180,E1 -11314.487,E2 -11314.487} C_VEL
LIN {X 0,Y 397.086,Z 499.646,A -85,B 0,C 180,E1 -11318.181,E2 -11318.181} C_VEL
LIN {X 0,Y 397.152,Z 499.642,A -85,B 0,C 180,E1 -11321.426,E2 -11321.426} C_VEL
LIN {X 0,Y 397.174,Z 499.634,A -85,B 0,C 180,E1 -11324.608,E2 -11324.608} C_VEL
LIN {X 0,Y 397.219,Z 499.633,A -85,B 0,C 180,E1 -11327.742,E2 -11327.742} C_VEL
LIN {X 0,Y 397.385,Z 499.609,A -85,B 0,C 180,E1 -11332.041,E2 -11332.041} C_VEL
LIN {X 0,Y 397.25,Z 499.625,A -85,B 0,C 180,E1 -11334.925,E2 -11334.925} C_VEL
LIN {X 0,Y 397.442,Z 499.603,A -85,B 0,C 180,E1 -11337.974,E2 -11337.974} C_VEL
LIN {X 0,Y 397.573,Z 499.586,A -85,B 0,C 180,E1 -11340,E2 -11340} C_VEL
LIN {X 0,Y 397.376,Z 499.611,A -85,B 0,C 180,E1 -11343.042,E2 -11343.042} C_VEL
LIN {X 0,Y 397.346,Z 499.612,A -85,B 0,C 180,E1 -11346.588,E2 -11346.588} C_VEL
LIN {X 0,Y 397.244,Z 499.628,A -85,B 0,C 180,E1 -11349.162,E2 -11349.162} C_VEL
LIN {X 0,Y 397.211,Z 499.63,A -85,B 0,C 180,E1 -11352.259,E2 -11352.259} C_VEL
LIN {X 0,Y 397.17,Z 499.639,A -85,B 0,C 180,E1 -11355.393,E2 -11355.393} C_VEL
LIN {X 0,Y 397.154,Z 499.636,A -85,B 0,C 180,E1 -11358.574,E2 -11358.574} C_VEL
LIN {X 0,Y 397.089,Z 499.649,A -85,B 0,C 180,E1 -11361.819,E2 -11361.819} C_VEL
LIN {X 0,Y 397.149,Z 499.639,A -85,B 0,C 180,E1 -11365.133,E2 -11365.133} C_VEL
LIN {X 0,Y 397.157,Z 499.64,A -85,B 0,C 180,E1 -11367.778,E2 -11367.778} C_VEL
LIN {X 0,Y 397.081,Z 499.646,A -85,B 0,C 180,E1 -11370.883,E2 -11370.883} C_VEL
LIN {X 0,Y 397.12,Z 499.641,A -85,B 0,C 180,E1 -11374.494,E2 -11374.494} C_VEL
LIN {X 0,Y 397.106,Z 499.643,A -85,B 0,C 180,E1 -11378.275,E2 -11378.275} C_VEL
LIN {X 0,Y 397.153,Z 499.639,A -85,B 0,C 180,E1 -11381.995,E2 -11381.995} C_VEL
LIN {X 0,Y 397.147,Z 499.639,A -85,B 0,C 180,E1 -11385.061,E2 -11385.061} C_VEL
LIN {X 0,Y 397.153,Z 499.639,A -85,B 0,C 180,E1 -11388.008,E2 -11388.008} C_VEL
LIN {X 0,Y 397.109,Z 499.647,A -85,B 0,C 180,E1 -11391.727,E2 -11391.727} C_VEL
LIN {X 0,Y 397.125,Z 499.645,A -85,B 0,C 180,E1 -11395.508,E2 -11395.508} C_VEL
LIN {X 0,Y 397.079,Z 499.648,A -85,B 0,C 180,E1 -11399.119,E2 -11399.119} C_VEL
LIN {X 0,Y 397.196,Z 499.631,A -85,B 0,C 180,E1 -11402.611,E2 -11402.611} C_VEL
LIN {X 0,Y 397.135,Z 499.642,A -85,B 0,C 180,E1 -11405.983,E2 -11405.983} C_VEL
LIN {X 0,Y 397.141,Z 499.643,A -85,B 0,C 180,E1 -11409.706,E2 -11409.706} C_VEL
LIN {X 0,Y 397.185,Z 499.633,A -85,B 0,C 180,E1 -11412.846,E2 -11412.846} C_VEL
LIN {X 0,Y 397.232,Z 499.627,A -85,B 0,C 180,E1 -11416.704,E2 -11416.704} C_VEL
LIN {X 0,Y 397.221,Z 499.632,A -85,B 0,C 180,E1 -11419.81,E2 -11419.81} C_VEL
LIN {X 0,Y 397.343,Z 499.613,A -85,B 0,C 180,E1 -11422.888,E2 -11422.888} C_VEL
LIN {X 0,Y 397.26,Z 499.624,A -85,B 0,C 180,E1 -11424.926,E2 -11424.926} C_VEL
LIN {X 0,Y 397.458,Z 499.602,A -85,B 0,C 180,E1 -11427.974,E2 -11427.974} C_VEL
LIN {X 0,Y 397.583,Z 499.586,A -85,B 0,C 180,E1 -11430.001,E2 -11430.001} C_VEL
LIN {X 0,Y 397.372,Z 499.612,A -85,B 0,C 180,E1 -11432.028,E2 -11432.028} C_VEL
LIN {X 0,Y 396.842,Z 499.679,A -85,B 0,C 180,E1 -11436.1,E2 -11436.1} C_VEL
LIN {X 0,Y 396.724,Z 499.703,A -85,B 0,C 180,E1 -11437.227,E2 -11437.227} C_VEL
LIN {X 0,Y 396.504,Z 502.158,A -85,B 0,C 180,E1 -11440.21,E2 -11440.21} C_VEL
LIN {X 0,Y 396.386,Z 504.767,A -85,B 0,C 180,E1 -11443.326,E2 -11443.326} C_VEL
LIN {X 0,Y 396.391,Z 505.821,A -85,B 0,C 180,E1 -11444.34,E2 -11444.34} C_VEL
LIN {X 0,Y 399.282,Z 513.904,A -85,B 0,C 180,E1 -11444.738,E2 -11444.738} C_VEL
LIN {X 0,Y 404.165,Z 528.288,A -85,B 0,C 180,E1 -11445.564,E2 -11445.564} C_VEL
LIN {X 0,Y 407.372,Z 539.664,A -85,B 0,C 180,E1 -11446.313,E2 -11446.313} C_VEL
LIN {X 0,Y 406.419,Z 554.435,A -85,B 0,C 180,E1 -11447.161,E2 -11447.161} C_VEL
LIN {X 0,Y 405.43,Z 559.796,A -85,B 0,C 180,E1 -11447.487,E2 -11447.487} C_VEL
LIN {X 0,Y 401.92,Z 568.4,A -85,B 0,C 180,E1 -11447.978,E2 -11447.978} C_VEL
LIN {X 0,Y 398.293,Z 576.786,A -85,B 0,C 180,E1 -11448.543,E2 -11448.543} C_VEL
LIN {X 0,Y 397.137,Z 581.678,A -85,B 0,C 180,E1 -11448.98,E2 -11448.98} C_VEL
LIN {X 0,Y 395.85,Z 593.744,A -85,B 0,C 180,E1 -11450.308,E2 -11450.308} C_VEL
LIN {X 0,Y 394.427,Z 604.441,A -85,B 0,C 180,E1 -11451.699,E2 -11451.699} C_VEL
LIN {X 0,Y 393.064,Z 615.516,A -85,B 0,C 180,E1 -11453.435,E2 -11453.435} C_VEL
LIN {X 0,Y 391.883,Z 624.919,A -85,B 0,C 180,E1 -11455.21,E2 -11455.21} C_VEL
LIN {X 0,Y 390.934,Z 632.809,A -85,B 0,C 180,E1 -11456.996,E2 -11456.996} C_VEL
LIN {X 0,Y 390.304,Z 638.596,A -85,B 0,C 180,E1 -11458.565,E2 -11458.565} C_VEL
LIN {X 0,Y 389.738,Z 644.035,A -85,B 0,C 180,E1 -11460.326,E2 -11460.326} C_VEL
LIN {X 0,Y 389.339,Z 648.186,A -85,B 0,C 180,E1 -11461.961,E2 -11461.961} C_VEL
LIN {X 0,Y 388.978,Z 652.284,A -85,B 0,C 180,E1 -11464.063,E2 -11464.063} C_VEL
LIN {X 0,Y 388.781,Z 654.473,A -85,B 0,C 180,E1 -11465.563,E2 -11465.563} C_VEL
LIN {X 0,Y 388.621,Z 656.639,A -85,B 0,C 180,E1 -11467.942,E2 -11467.942} C_VEL
LIN {X 0,Y 388.569,Z 657.188,A -85,B 0,C 180,E1 -11469.275,E2 -11469.275} C_VEL
LIN {X 0,Y 388.574,Z 657.276,A -85,B 0,C 180,E1 -11470.626,E2 -11470.626} C_VEL
LIN {X 0,Y 388.617,Z 656.827,A -85,B 0,C 180,E1 -11472.142,E2 -11472.142} C_VEL
LIN {X 0,Y 388.717,Z 655.76,A -85,B 0,C 180,E1 -11473.68,E2 -11473.68} C_VEL
LIN {X 0,Y 388.912,Z 654.049,A -85,B 0,C 180,E1 -11475.189,E2 -11475.189} C_VEL
LIN {X 0,Y 389.253,Z 650.762,A -85,B 0,C 180,E1 -11477.242,E2 -11477.242} C_VEL
LIN {X 0,Y 389.663,Z 646.397,A -85,B 0,C 180,E1 -11479.245,E2 -11479.245} C_VEL
LIN {X 0,Y 390.342,Z 640.667,A -85,B 0,C 180,E1 -11481.268,E2 -11481.268} C_VEL
LIN {X 0,Y 391.23,Z 633.355,A -85,B 0,C 180,E1 -11483.326,E2 -11483.326} C_VEL
LIN {X 0,Y 392.392,Z 624.743,A -85,B 0,C 180,E1 -11485.286,E2 -11485.286} C_VEL
LIN {X 0,Y 393.636,Z 615.357,A -85,B 0,C 180,E1 -11487.049,E2 -11487.049} C_VEL
LIN {X 0,Y 395.132,Z 604.397,A -85,B 0,C 180,E1 -11488.756,E2 -11488.756} C_VEL
LIN {X 0,Y 396.647,Z 592.787,A -85,B 0,C 180,E1 -11490.256,E2 -11490.256} C_VEL
LIN {X 0,Y 398.216,Z 579.793,A -85,B 0,C 180,E1 -11491.645,E2 -11491.645} C_VEL
LIN {X 0,Y 399.76,Z 565.227,A -85,B 0,C 180,E1 -11492.902,E2 -11492.902} C_VEL
LIN {X 0,Y 401.072,Z 551.72,A -85,B 0,C 180,E1 -11493.83,E2 -11493.83} C_VEL
LIN {X 0,Y 401.591,Z 541.895,A -85,B 0,C 180,E1 -11494.394,E2 -11494.394} C_VEL
LIN {X 0,Y 397.307,Z 528,A -85,B 0,C 180,E1 -11495.402,E2 -11495.402} C_VEL
LIN {X 0,Y 392.066,Z 514.637,A -85,B 0,C 180,E1 -11496.304,E2 -11496.304} C_VEL
LIN {X 0,Y 389.68,Z 509.049,A -85,B 0,C 180,E1 -11496.65,E2 -11496.65} C_VEL
LIN {X 0,Y 389.569,Z 508.269,A -85,B 0,C 180,E1 -11496.724,E2 -11496.724} C_VEL
LIN {X 0,Y 389.718,Z 505.925,A -85,B 0,C 180,E1 -11499.962,E2 -11499.962} C_VEL
LIN {X 0,Y 389.859,Z 503.63,A -85,B 0,C 180,E1 -11503.235,E2 -11503.235} C_VEL
LIN {X 0,Y 390.022,Z 501.295,A -85,B 0,C 180,E1 -11506.666,E2 -11506.666} C_VEL
LIN {X 0,Y 390.026,Z 500.754,A -85,B 0,C 180,E1 -11507.512,E2 -11507.512} C_VEL
LIN {X 0,Y 390.197,Z 500.507,A -85,B 0,C 180,E1 -11510.671,E2 -11510.671} C_VEL
LIN {X 0,Y 390.325,Z 500.492,A -85,B 0,C 180,E1 -11513.798,E2 -11513.798} C_VEL
LIN {X 0,Y 390.418,Z 500.479,A -85,B 0,C 180,E1 -11517.936,E2 -11517.936} C_VEL
LIN {X 0,Y 390.547,Z 500.462,A -85,B 0,C 180,E1 -11520,E2 -11520} C_VEL
LIN {X 0,Y 390.312,Z 500.492,A -85,B 0,C 180,E1 -11523.096,E2 -11523.096} C_VEL
LIN {X 0,Y 390.328,Z 500.489,A -85,B 0,C 180,E1 -11526.202,E2 -11526.202} C_VEL
LIN {X 0,Y 390.312,Z 500.491,A -85,B 0,C 180,E1 -11528.282,E2 -11528.282} C_VEL
LIN {X 0,Y 390.168,Z 500.51,A -85,B 0,C 180,E1 -11532.483,E2 -11532.483} C_VEL
LIN {X 0,Y 390.135,Z 500.511,A -85,B 0,C 180,E1 -11535.677,E2 -11535.677} C_VEL
LIN {X 0,Y 390.102,Z 500.516,A -85,B 0,C 180,E1 -11538.922,E2 -11538.922} C_VEL
LIN {X 0,Y 390.037,Z 500.527,A -85,B 0,C 180,E1 -11542.234,E2 -11542.234} C_VEL
LIN {X 0,Y 390.116,Z 500.516,A -85,B 0,C 180,E1 -11545.743,E2 -11545.743} C_VEL
LIN {X 0,Y 390.062,Z 500.523,A -85,B 0,C 180,E1 -11549.109,E2 -11549.109} C_VEL
LIN {X 0,Y 390.041,Z 500.526,A -85,B 0,C 180,E1 -11552.721,E2 -11552.721} C_VEL
LIN {X 0,Y 390.054,Z 500.524,A -85,B 0,C 180,E1 -11555.825,E2 -11555.825} C_VEL
LIN {X 0,Y 390.084,Z 500.76,A -85,B 0,C 180,E1 -11556.762,E2 -11556.762} C_VEL
LIN {X 0,Y 390.636,Z 503.58,A -85,B 0,C 180,E1 -11559.32,E2 -11559.32} C_VEL
LIN {X 0,Y 391.313,Z 507.659,A -85,B 0,C 180,E1 -11562.578,E2 -11562.578} C_VEL
LIN {X 0,Y 392.1,Z 512.189,A -85,B 0,C 180,E1 -11565.804,E2 -11565.804} C_VEL
LIN {X 0,Y 392.45,Z 515.371,A -85,B 0,C 180,E1 -11567.884,E2 -11567.884} C_VEL
LIN {X 0,Y 391.897,Z 520.946,A -85,B 0,C 180,E1 -11571.122,E2 -11571.122} C_VEL
LIN {X 0,Y 391.474,Z 525.957,A -85,B 0,C 180,E1 -11573.888,E2 -11573.888} C_VEL
LIN {X 0,Y 390.935,Z 531.45,A -85,B 0,C 180,E1 -11576.749,E2 -11576.749} C_VEL
LIN {X 0,Y 390.507,Z 537.475,A -85,B 0,C 180,E1 -11579.752,E2 -11579.752} C_VEL
LIN {X 0,Y 390.018,Z 544.964,A -85,B 0,C 180,E1 -11583.337,E2 -11583.337} C_VEL
LIN {X 0,Y 390.8,Z 548.09,A -85,B 0,C 180,E1 -11583.472,E2 -11583.472} C_VEL
LIN {X 0,Y 395.148,Z 564.237,A -85,B 0,C 180,E1 -11584.292,E2 -11584.292} C_VEL
LIN {X 0,Y 398.064,Z 578.716,A -85,B 0,C 180,E1 -11585.133,E2 -11585.133} C_VEL
LIN {X 0,Y 399.905,Z 592.448,A -85,B 0,C 180,E1 -11586.043,E2 -11586.043} C_VEL
LIN {X 0,Y 398.4,Z 607.696,A -85,B 0,C 180,E1 -11587.053,E2 -11587.053} C_VEL
LIN {X 0,Y 396.897,Z 621.108,A -85,B 0,C 180,E1 -11588.17,E2 -11588.17} C_VEL
LIN {X 0,Y 395.323,Z 633.749,A -85,B 0,C 180,E1 -11589.444,E2 -11589.444} C_VEL
LIN {X 0,Y 393.897,Z 645.54,A -85,B 0,C 180,E1 -11590.875,E2 -11590.875} C_VEL
LIN {X 0,Y 392.488,Z 657.046,A -85,B 0,C 180,E1 -11592.546,E2 -11592.546} C_VEL
LIN {X 0,Y 391.369,Z 666.087,A -85,B 0,C 180,E1 -11594.106,E2 -11594.106} C_VEL
LIN {X 0,Y 390.416,Z 675.025,A -85,B 0,C 180,E1 -11595.935,E2 -11595.935} C_VEL
LIN {X 0,Y 389.807,Z 681.523,A -85,B 0,C 180,E1 -11597.505,E2 -11597.505} C_VEL
LIN {X 0,Y 389.178,Z 688.668,A -85,B 0,C 180,E1 -11599.596,E2 -11599.596} C_VEL
LIN {X 0,Y 388.935,Z 694.319,A -85,B 0,C 180,E1 -11601.688,E2 -11601.688} C_VEL
LIN {X 0,Y 388.775,Z 698.74,A -85,B 0,C 180,E1 -11603.851,E2 -11603.851} C_VEL
LIN {X 0,Y 388.72,Z 701.607,A -85,B 0,C 180,E1 -11605.852,E2 -11605.852} C_VEL
LIN {X 0,Y 388.83,Z 703.417,A -85,B 0,C 180,E1 -11607.928,E2 -11607.928} C_VEL
LIN {X 0,Y 388.808,Z 704.047,A -85,B 0,C 180,E1 -11609.999,E2 -11609.999} C_VEL
LIN {X 0,Y 388.829,Z 703.46,A -85,B 0,C 180,E1 -11612.071,E2 -11612.071} C_VEL
LIN {X 0,Y 388.714,Z 701.665,A -85,B 0,C 180,E1 -11614.147,E2 -11614.147} C_VEL
LIN {X 0,Y 388.831,Z 698.675,A -85,B 0,C 180,E1 -11616.225,E2 -11616.225} C_VEL
LIN {X 0,Y 388.938,Z 694.401,A -85,B 0,C 180,E1 -11618.311,E2 -11618.311} C_VEL
LIN {X 0,Y 389.178,Z 688.737,A -85,B 0,C 180,E1 -11620.403,E2 -11620.403} C_VEL
LIN {X 0,Y 389.794,Z 681.549,A -85,B 0,C 180,E1 -11622.495,E2 -11622.495} C_VEL
LIN {X 0,Y 390.521,Z 673.859,A -85,B 0,C 180,E1 -11624.326,E2 -11624.326} C_VEL
LIN {X 0,Y 391.497,Z 664.608,A -85,B 0,C 180,E1 -11626.155,E2 -11626.155} C_VEL
LIN {X 0,Y 392.718,Z 655.186,A -85,B 0,C 180,E1 -11627.711,E2 -11627.711} C_VEL
LIN {X 0,Y 394.068,Z 643.348,A -85,B 0,C 180,E1 -11629.359,E2 -11629.359} C_VEL
LIN {X 0,Y 395.569,Z 630.684,A -85,B 0,C 180,E1 -11630.813,E2 -11630.813} C_VEL
LIN {X 0,Y 397.089,Z 617.099,A -85,B 0,C 180,E1 -11632.091,E2 -11632.091} C_VEL
LIN {X 0,Y 398.71,Z 602.2,A -85,B 0,C 180,E1 -11633.208,E2 -11633.208} C_VEL
LIN {X 0,Y 399.49,Z 591.508,A -85,B 0,C 180,E1 -11633.867,E2 -11633.867} C_VEL
LIN {X 0,Y 396.922,Z 576.132,A -85,B 0,C 180,E1 -11634.825,E2 -11634.825} C_VEL
LIN {X 0,Y 393.609,Z 560.94,A -85,B 0,C 180,E1 -11635.613,E2 -11635.613} C_VEL
LIN {X 0,Y 390.057,Z 547.037,A -85,B 0,C 180,E1 -11636.229,E2 -11636.229} C_VEL
LIN {X 0,Y 390.532,Z 539.834,A -85,B 0,C 180,E1 -11639.661,E2 -11639.661} C_VEL
LIN {X 0,Y 391.157,Z 532.57,A -85,B 0,C 180,E1 -11643.229,E2 -11643.229} C_VEL
LIN {X 0,Y 391.579,Z 526.484,A -85,B 0,C 180,E1 -11646.317,E2 -11646.317} C_VEL
LIN {X 0,Y 392.253,Z 520.233,A -85,B 0,C 180,E1 -11649.608,E2 -11649.608} C_VEL
LIN {X 0,Y 392.557,Z 515.692,A -85,B 0,C 180,E1 -11652.115,E2 -11652.115} C_VEL
LIN {X 0,Y 392.133,Z 511.905,A -85,B 0,C 180,E1 -11654.343,E2 -11654.343} C_VEL
LIN {X 0,Y 391.214,Z 507.009,A -85,B 0,C 180,E1 -11657.436,E2 -11657.436} C_VEL
LIN {X 0,Y 390.311,Z 501.781,A -85,B 0,C 180,E1 -11660.934,E2 -11660.934} C_VEL
LIN {X 0,Y 390.06,Z 500.525,A -85,B 0,C 180,E1 -11661.895,E2 -11661.895} C_VEL
LIN {X 0,Y 390.077,Z 500.52,A -85,B 0,C 180,E1 -11664.793,E2 -11664.793} C_VEL
LIN {X 0,Y 390.018,Z 500.525,A -85,B 0,C 180,E1 -11668.496,E2 -11668.496} C_VEL
LIN {X 0,Y 390.108,Z 500.515,A -85,B 0,C 180,E1 -11672.07,E2 -11672.07} C_VEL
LIN {X 0,Y 390.068,Z 500.524,A -85,B 0,C 180,E1 -11675.519,E2 -11675.519} C_VEL
LIN {X 0,Y 390.077,Z 500.523,A -85,B 0,C 180,E1 -11679.53,E2 -11679.53} C_VEL
LIN {X 0,Y 390.131,Z 500.515,A -85,B 0,C 180,E1 -11683.248,E2 -11683.248} C_VEL
LIN {X 0,Y 390.184,Z 500.504,A -85,B 0,C 180,E1 -11686.561,E2 -11686.561} C_VEL
LIN {X 0,Y 390.169,Z 500.511,A -85,B 0,C 180,E1 -11689.623,E2 -11689.623} C_VEL
LIN {X 0,Y 390.309,Z 500.489,A -85,B 0,C 180,E1 -11692.759,E2 -11692.759} C_VEL
LIN {X 0,Y 390.221,Z 500.5,A -85,B 0,C 180,E1 -11694.834,E2 -11694.834} C_VEL
LIN {X 0,Y 390.411,Z 500.479,A -85,B 0,C 180,E1 -11697.937,E2 -11697.937} C_VEL
LIN {X 0,Y 390.542,Z 500.462,A -85,B 0,C 180,E1 -11700,E2 -11700} C_VEL
LIN {X 0,Y 390.31,Z 500.491,A -85,B 0,C 180,E1 -11703.097,E2 -11703.097} C_VEL
LIN {X 0,Y 390.302,Z 500.489,A -85,B 0,C 180,E1 -11706.581,E2 -11706.581} C_VEL
LIN {X 0,Y 390.196,Z 500.507,A -85,B 0,C 180,E1 -11709.329,E2 -11709.329} C_VEL
LIN {X 0,Y 390.162,Z 500.507,A -85,B 0,C 180,E1 -11712.484,E2 -11712.484} C_VEL
LIN {X 0,Y 390.13,Z 500.516,A -85,B 0,C 180,E1 -11715.678,E2 -11715.678} C_VEL
LIN {X 0,Y 390.097,Z 500.516,A -85,B 0,C 180,E1 -11718.923,E2 -11718.923} C_VEL
LIN {X 0,Y 390.032,Z 500.524,A -85,B 0,C 180,E1 -11722.235,E2 -11722.235} C_VEL
LIN {X 0,Y 390.112,Z 500.518,A -85,B 0,C 180,E1 -11725.744,E2 -11725.744} C_VEL
LIN {X 0,Y 390.059,Z 500.522,A -85,B 0,C 180,E1 -11729.11,E2 -11729.11} C_VEL
LIN {X 0,Y 390.05,Z 500.521,A -85,B 0,C 180,E1 -11732.721,E2 -11732.721} C_VEL
LIN {X 0,Y 390.052,Z 500.525,A -85,B 0,C 180,E1 -11735.827,E2 -11735.827} C_VEL
LIN {X 0,Y 390.071,Z 500.521,A -85,B 0,C 180,E1 -11739.221,E2 -11739.221} C_VEL
LIN {X 0,Y 390.119,Z 500.513,A -85,B 0,C 180,E1 -11742.388,E2 -11742.388} C_VEL
LIN {X 0,Y 390.114,Z 500.518,A -85,B 0,C 180,E1 -11745.366,E2 -11745.366} C_VEL
LIN {X 0,Y 390.102,Z 500.515,A -85,B 0,C 180,E1 -11748.198,E2 -11748.198} C_VEL
LIN {X 0,Y 390.094,Z 500.516,A -85,B 0,C 180,E1 -11750.91,E2 -11750.91} C_VEL
LIN {X 0,Y 390.085,Z 500.517,A -85,B 0,C 180,E1 -11754.795,E2 -11754.795} C_VEL
LIN {X 0,Y 390.023,Z 500.524,A -85,B 0,C 180,E1 -11758.497,E2 -11758.497} C_VEL
LIN {X 0,Y 390.118,Z 500.514,A -85,B 0,C 180,E1 -11762.071,E2 -11762.071} C_VEL
LIN {X 0,Y 390.083,Z 500.522,A -85,B 0,C 180,E1 -11765.521,E2 -11765.521} C_VEL
LIN {X 0,Y 390.058,Z 500.521,A -85,B 0,C 180,E1 -11768.879,E2 -11768.879} C_VEL
LIN {X 0,Y 390.131,Z 500.512,A -85,B 0,C 180,E1 -11772.168,E2 -11772.168} C_VEL
LIN {X 0,Y 390.148,Z 500.513,A -85,B 0,C 180,E1 -11775.394,E2 -11775.394} C_VEL
LIN {X 0,Y 390.151,Z 500.508,A -85,B 0,C 180,E1 -11778.572,E2 -11778.572} C_VEL
LIN {X 0,Y 390.274,Z 500.495,A -85,B 0,C 180,E1 -11782.072,E2 -11782.072} C_VEL
LIN {X 0,Y 390.231,Z 500.499,A -85,B 0,C 180,E1 -11784.834,E2 -11784.834} C_VEL
LIN {X 0,Y 390.426,Z 500.478,A -85,B 0,C 180,E1 -11787.937,E2 -11787.937} C_VEL
LIN {X 0,Y 390.552,Z 500.461,A -85,B 0,C 180,E1 -11790.001,E2 -11790.001} C_VEL
LIN {X 0,Y 390.332,Z 500.489,A -85,B 0,C 180,E1 -11792.064,E2 -11792.064} C_VEL
LIN {X 0,Y 389.94,Z 500.538,A -85,B 0,C 180,E1 -11795.171,E2 -11795.171} C_VEL
LIN {X 0,Y 389.683,Z 500.576,A -85,B 0,C 180,E1 -11797.277,E2 -11797.277} C_VEL
LIN {X 0,Y 389.438,Z 503.14,A -85,B 0,C 180,E1 -11800.397,E2 -11800.397} C_VEL
LIN {X 0,Y 389.339,Z 505.989,A -85,B 0,C 180,E1 -11803.838,E2 -11803.838} C_VEL
LIN {X 0,Y 391.716,Z 512.81,A -85,B 0,C 180,E1 -11804.199,E2 -11804.199} C_VEL
LIN {X 0,Y 396.866,Z 527.572,A -85,B 0,C 180,E1 -11805.066,E2 -11805.066} C_VEL
LIN {X 0,Y 400.569,Z 540.33,A -85,B 0,C 180,E1 -11805.927,E2 -11805.927} C_VEL
LIN {X 0,Y 400.712,Z 543.446,A -85,B 0,C 180,E1 -11806.106,E2 -11806.106} C_VEL
LIN {X 0,Y 399.54,Z 558.109,A -85,B 0,C 180,E1 -11807.004,E2 -11807.004} C_VEL
LIN {X 0,Y 398.182,Z 572.217,A -85,B 0,C 180,E1 -11808.098,E2 -11808.098} C_VEL
LIN {X 0,Y 397.137,Z 581.678,A -85,B 0,C 180,E1 -11808.98,E2 -11808.98} C_VEL
LIN {X 0,Y 395.988,Z 586.536,A -85,B 0,C 180,E1 -11809.445,E2 -11809.445} C_VEL
LIN {X 0,Y 392.333,Z 594.259,A -85,B 0,C 180,E1 -11810.176,E2 -11810.176} C_VEL
LIN {X 0,Y 388.657,Z 601.682,A -85,B 0,C 180,E1 -11810.981,E2 -11810.981} C_VEL
LIN {X 0,Y 387.492,Z 605.934,A -85,B 0,C 180,E1 -11811.557,E2 -11811.557} C_VEL
LIN {X 0,Y 386.118,Z 616.818,A -85,B 0,C 180,E1 -11813.321,E2 -11813.321} C_VEL
LIN {X 0,Y 384.872,Z 626.061,A -85,B 0,C 180,E1 -11815.123,E2 -11815.123} C_VEL
LIN {X 0,Y 384.008,Z 633.046,A -85,B 0,C 180,E1 -11816.737,E2 -11816.737} C_VEL
LIN {X 0,Y 383.287,Z 639.329,A -85,B 0,C 180,E1 -11818.473,E2 -11818.473} C_VEL
LIN {X 0,Y 382.664,Z 644.86,A -85,B 0,C 180,E1 -11820.321,E2 -11820.321} C_VEL
LIN {X 0,Y 382.221,Z 649.478,A -85,B 0,C 180,E1 -11822.24,E2 -11822.24} C_VEL
LIN {X 0,Y 381.891,Z 652.904,A -85,B 0,C 180,E1 -11824.091,E2 -11824.091} C_VEL
LIN {X 0,Y 381.624,Z 655.552,A -85,B 0,C 180,E1 -11826.108,E2 -11826.108} C_VEL
LIN {X 0,Y 381.534,Z 656.875,A -85,B 0,C 180,E1 -11827.619,E2 -11827.619} C_VEL
LIN {X 0,Y 381.486,Z 657.62,A -85,B 0,C 180,E1 -11829.307,E2 -11829.307} C_VEL
LIN {X 0,Y 381.494,Z 657.533,A -85,B 0,C 180,E1 -11831.544,E2 -11831.544} C_VEL
LIN {X 0,Y 381.59,Z 656.804,A -85,B 0,C 180,E1 -11832.957,E2 -11832.957} C_VEL
LIN {X 0,Y 381.736,Z 655.556,A -85,B 0,C 180,E1 -11834.395,E2 -11834.395} C_VEL
LIN {X 0,Y 382.076,Z 652.768,A -85,B 0,C 180,E1 -11836.486,E2 -11836.486} C_VEL
LIN {X 0,Y 382.476,Z 648.785,A -85,B 0,C 180,E1 -11838.585,E2 -11838.585} C_VEL
LIN {X 0,Y 382.945,Z 644.262,A -85,B 0,C 180,E1 -11840.426,E2 -11840.426} C_VEL
LIN {X 0,Y 383.748,Z 638.089,A -85,B 0,C 180,E1 -11842.413,E2 -11842.413} C_VEL
LIN {X 0,Y 384.838,Z 630.129,A -85,B 0,C 180,E1 -11844.485,E2 -11844.485} C_VEL
LIN {X 0,Y 385.967,Z 621.935,A -85,B 0,C 180,E1 -11846.24,E2 -11846.24} C_VEL
LIN {X 0,Y 387.359,Z 612.411,A -85,B 0,C 180,E1 -11847.947,E2 -11847.947} C_VEL
LIN {X 0,Y 388.968,Z 601.282,A -85,B 0,C 180,E1 -11849.607,E2 -11849.607} C_VEL
LIN {X 0,Y 390.462,Z 589.842,A -85,B 0,C 180,E1 -11851.033,E2 -11851.033} C_VEL
LIN {X 0,Y 392.069,Z 576.933,A -85,B 0,C 180,E1 -11852.361,E2 -11852.361} C_VEL
LIN {X 0,Y 393.511,Z 563.634,A -85,B 0,C 180,E1 -11853.481,E2 -11853.481} C_VEL
LIN {X 0,Y 394.953,Z 548.832,A -85,B 0,C 180,E1 -11854.465,E2 -11854.465} C_VEL
LIN {X 0,Y 395.254,Z 544.121,A -85,B 0,C 180,E1 -11854.738,E2 -11854.738} C_VEL
LIN {X 0,Y 390.983,Z 529.992,A -85,B 0,C 180,E1 -11855.817,E2 -11855.817} C_VEL
LIN {X 0,Y 385.945,Z 517.173,A -85,B 0,C 180,E1 -11856.729,E2 -11856.729} C_VEL
LIN {X 0,Y 382.672,Z 509.572,A -85,B 0,C 180,E1 -11857.227,E2 -11857.227} C_VEL
LIN {X 0,Y 382.542,Z 508.795,A -85,B 0,C 180,E1 -11857.306,E2 -11857.306} C_VEL
LIN {X 0,Y 382.691,Z 506.387,A -85,B 0,C 180,E1 -11860.696,E2 -11860.696} C_VEL
LIN {X 0,Y 382.864,Z 504.118,A -85,B 0,C 180,E1 -11864.017,E2 -11864.017} C_VEL
LIN {X 0,Y 383.011,Z 501.986,A -85,B 0,C 180,E1 -11867.279,E2 -11867.279} C_VEL
LIN {X 0,Y 382.999,Z 501.408,A -85,B 0,C 180,E1 -11868.354,E2 -11868.354} C_VEL
LIN {X 0,Y 383.263,Z 501.371,A -85,B 0,C 180,E1 -11871.974,E2 -11871.974} C_VEL
LIN {X 0,Y 383.198,Z 501.378,A -85,B 0,C 180,E1 -11874.738,E2 -11874.738} C_VEL
LIN {X 0,Y 383.385,Z 501.355,A -85,B 0,C 180,E1 -11877.898,E2 -11877.898} C_VEL
LIN {X 0,Y 383.516,Z 501.338,A -85,B 0,C 180,E1 -11880,E2 -11880} C_VEL
LIN {X 0,Y 383.249,Z 501.371,A -85,B 0,C 180,E1 -11883.153,E2 -11883.153} C_VEL
LIN {X 0,Y 383.285,Z 501.366,A -85,B 0,C 180,E1 -11886.316,E2 -11886.316} C_VEL
LIN {X 0,Y 383.257,Z 501.37,A -85,B 0,C 180,E1 -11888.435,E2 -11888.435} C_VEL
LIN {X 0,Y 383.095,Z 501.389,A -85,B 0,C 180,E1 -11891.642,E2 -11891.642} C_VEL
LIN {X 0,Y 383.106,Z 501.388,A -85,B 0,C 180,E1 -11894.881,E2 -11894.881} C_VEL
LIN {X 0,Y 383.086,Z 501.391,A -85,B 0,C 180,E1 -11898.172,E2 -11898.172} C_VEL
LIN {X 0,Y 382.99,Z 501.401,A -85,B 0,C 180,E1 -11901.531,E2 -11901.531} C_VEL
LIN {X 0,Y 383.049,Z 501.394,A -85,B 0,C 180,E1 -11904.96,E2 -11904.96} C_VEL
LIN {X 0,Y 383.047,Z 501.396,A -85,B 0,C 180,E1 -11908.492,E2 -11908.492} C_VEL
LIN {X 0,Y 383.008,Z 501.403,A -85,B 0,C 180,E1 -11912.149,E2 -11912.149} C_VEL
LIN {X 0,Y 383.028,Z 501.399,A -85,B 0,C 180,E1 -11915.853,E2 -11915.853} C_VEL
LIN {X 0,Y 383.517,Z 504.199,A -85,B 0,C 180,E1 -11918.539,E2 -11918.539} C_VEL
LIN {X 0,Y 384.097,Z 507.592,A -85,B 0,C 180,E1 -11921.393,E2 -11921.393} C_VEL
LIN {X 0,Y 384.809,Z 511.801,A -85,B 0,C 180,E1 -11924.58,E2 -11924.58} C_VEL
LIN {X 0,Y 385.442,Z 516.167,A -85,B 0,C 180,E1 -11927.574,E2 -11927.574} C_VEL
LIN {X 0,Y 385.036,Z 520.674,A -85,B 0,C 180,E1 -11930.294,E2 -11930.294} C_VEL
LIN {X 0,Y 384.389,Z 527.593,A -85,B 0,C 180,E1 -11934.192,E2 -11934.192} C_VEL
LIN {X 0,Y 383.815,Z 533.638,A -85,B 0,C 180,E1 -11937.384,E2 -11937.384} C_VEL
LIN {X 0,Y 383.357,Z 539.482,A -85,B 0,C 180,E1 -11940.331,E2 -11940.331} C_VEL
LIN {X 0,Y 383.015,Z 544.411,A -85,B 0,C 180,E1 -11942.741,E2 -11942.741} C_VEL
LIN {X 0,Y 383.904,Z 547.804,A -85,B 0,C 180,E1 -11942.914,E2 -11942.914} C_VEL
LIN {X 0,Y 388.177,Z 563.098,A -85,B 0,C 180,E1 -11943.728,E2 -11943.728} C_VEL
LIN {X 0,Y 391.266,Z 578.257,A -85,B 0,C 180,E1 -11944.641,E2 -11944.641} C_VEL
LIN {X 0,Y 393.309,Z 593.558,A -85,B 0,C 180,E1 -11945.687,E2 -11945.687} C_VEL
LIN {X 0,Y 391.842,Z 607.684,A -85,B 0,C 180,E1 -11946.655,E2 -11946.655} C_VEL
LIN {X 0,Y 390.253,Z 620.919,A -85,B 0,C 180,E1 -11947.779,E2 -11947.779} C_VEL
LIN {X 0,Y 388.477,Z 634.669,A -85,B 0,C 180,E1 -11949.204,E2 -11949.204} C_VEL
LIN {X 0,Y 387.01,Z 646.107,A -85,B 0,C 180,E1 -11950.645,E2 -11950.645} C_VEL
LIN {X 0,Y 385.634,Z 656.693,A -85,B 0,C 180,E1 -11952.226,E2 -11952.226} C_VEL
LIN {X 0,Y 384.459,Z 665.719,A -85,B 0,C 180,E1 -11953.813,E2 -11953.813} C_VEL
LIN {X 0,Y 383.448,Z 674.645,A -85,B 0,C 180,E1 -11955.674,E2 -11955.674} C_VEL
LIN {X 0,Y 382.788,Z 681.141,A -85,B 0,C 180,E1 -11957.272,E2 -11957.272} C_VEL
LIN {X 0,Y 382.135,Z 688.277,A -85,B 0,C 180,E1 -11959.402,E2 -11959.402} C_VEL
LIN {X 0,Y 381.869,Z 693.912,A -85,B 0,C 180,E1 -11961.533,E2 -11961.533} C_VEL
LIN {X 0,Y 381.68,Z 698.591,A -85,B 0,C 180,E1 -11963.887,E2 -11963.887} C_VEL
LIN {X 0,Y 381.644,Z 701.189,A -85,B 0,C 180,E1 -11965.775,E2 -11965.775} C_VEL
LIN {X 0,Y 381.761,Z 702.994,A -85,B 0,C 180,E1 -11967.889,E2 -11967.889} C_VEL
LIN {X 0,Y 381.734,Z 703.617,A -85,B 0,C 180,E1 -11969.999,E2 -11969.999} C_VEL
LIN {X 0,Y 381.76,Z 703.028,A -85,B 0,C 180,E1 -11972.109,E2 -11972.109} C_VEL
LIN {X 0,Y 381.64,Z 701.225,A -85,B 0,C 180,E1 -11974.224,E2 -11974.224} C_VEL
LIN {X 0,Y 381.761,Z 698.224,A -85,B 0,C 180,E1 -11976.341,E2 -11976.341} C_VEL
LIN {X 0,Y 381.873,Z 693.936,A -85,B 0,C 180,E1 -11978.466,E2 -11978.466} C_VEL
LIN {X 0,Y 382.136,Z 688.259,A -85,B 0,C 180,E1 -11980.597,E2 -11980.597} C_VEL
LIN {X 0,Y 382.597,Z 683.02,A -85,B 0,C 180,E1 -11982.195,E2 -11982.195} C_VEL
LIN {X 0,Y 383.301,Z 675.678,A -85,B 0,C 180,E1 -11984.06,E2 -11984.06} C_VEL
LIN {X 0,Y 384.276,Z 666.863,A -85,B 0,C 180,E1 -11985.921,E2 -11985.921} C_VEL
LIN {X 0,Y 385.648,Z 656.272,A -85,B 0,C 180,E1 -11987.772,E2 -11987.772} C_VEL
LIN {X 0,Y 386.96,Z 645.405,A -85,B 0,C 180,E1 -11989.356,E2 -11989.356} C_VEL
LIN {X 0,Y 388.389,Z 633.574,A -85,B 0,C 180,E1 -11990.8,E2 -11990.8} C_VEL
LIN {X 0,Y 389.931,Z 620.688,A -85,B 0,C 180,E1 -11992.1,E2 -11992.1} C_VEL
LIN {X 0,Y 391.55,Z 606.541,A -85,B 0,C 180,E1 -11993.258,E2 -11993.258} C_VEL
LIN {X 0,Y 392.809,Z 592.982,A -85,B 0,C 180,E1 -11994.151,E2 -11994.151} C_VEL
LIN {X 0,Y 390.379,Z 577.861,A -85,B 0,C 180,E1 -11995.14,E2 -11995.14} C_VEL
LIN {X 0,Y 387.179,Z 562.866,A -85,B 0,C 180,E1 -11995.965,E2 -11995.965} C_VEL
LIN {X 0,Y 383.028,Z 546.675,A -85,B 0,C 180,E1 -11996.714,E2 -11996.714} C_VEL
LIN {X 0,Y 383.459,Z 540.59,A -85,B 0,C 180,E1 -11999.659,E2 -11999.659} C_VEL
LIN {X 0,Y 384.13,Z 533.333,A -85,B 0,C 180,E1 -12003.289,E2 -12003.289} C_VEL
LIN {X 0,Y 384.565,Z 527.219,A -85,B 0,C 180,E1 -12006.476,E2 -12006.476} C_VEL
LIN {X 0,Y 385.295,Z 520.672,A -85,B 0,C 180,E1 -12009.995,E2 -12009.995} C_VEL
LIN {X 0,Y 385.532,Z 516.399,A -85,B 0,C 180,E1 -12012.413,E2 -12012.413} C_VEL
LIN {X 0,Y 385.094,Z 512.75,A -85,B 0,C 180,E1 -12014.623,E2 -12014.623} C_VEL
LIN {X 0,Y 384.252,Z 508.401,A -85,B 0,C 180,E1 -12017.411,E2 -12017.411} C_VEL
LIN {X 0,Y 383.515,Z 504.092,A -85,B 0,C 180,E1 -12020.321,E2 -12020.321} C_VEL
LIN {X 0,Y 383.005,Z 501.402,A -85,B 0,C 180,E1 -12022.296,E2 -12022.296} C_VEL
LIN {X 0,Y 383.009,Z 501.403,A -85,B 0,C 180,E1 -12025.659,E2 -12025.659} C_VEL
LIN {X 0,Y 382.977,Z 501.404,A -85,B 0,C 180,E1 -12029.081,E2 -12029.081} C_VEL
LIN {X 0,Y 383.047,Z 501.393,A -85,B 0,C 180,E1 -12032.698,E2 -12032.698} C_VEL
LIN {X 0,Y 383.042,Z 501.396,A -85,B 0,C 180,E1 -12035.039,E2 -12035.039} C_VEL
LIN {X 0,Y 382.982,Z 501.401,A -85,B 0,C 180,E1 -12038.469,E2 -12038.469} C_VEL
LIN {X 0,Y 383.08,Z 501.392,A -85,B 0,C 180,E1 -12041.828,E2 -12041.828} C_VEL
LIN {X 0,Y 383.104,Z 501.388,A -85,B 0,C 180,E1 -12045.118,E2 -12045.118} C_VEL
LIN {X 0,Y 383.097,Z 501.387,A -85,B 0,C 180,E1 -12048.358,E2 -12048.358} C_VEL
LIN {X 0,Y 383.294,Z 501.365,A -85,B 0,C 180,E1 -12051.933,E2 -12051.933} C_VEL
LIN {X 0,Y 383.193,Z 501.375,A -85,B 0,C 180,E1 -12054.739,E2 -12054.739} C_VEL
LIN {X 0,Y 383.379,Z 501.355,A -85,B 0,C 180,E1 -12057.899,E2 -12057.899} C_VEL
LIN {X 0,Y 383.511,Z 501.337,A -85,B 0,C 180,E1 -12060,E2 -12060} C_VEL
LIN {X 0,Y 383.247,Z 501.371,A -85,B 0,C 180,E1 -12063.154,E2 -12063.154} C_VEL
LIN {X 0,Y 383.263,Z 501.366,A -85,B 0,C 180,E1 -12066.571,E2 -12066.571} C_VEL
LIN {X 0,Y 383.143,Z 501.387,A -85,B 0,C 180,E1 -12069.503,E2 -12069.503} C_VEL
LIN {X 0,Y 383.117,Z 501.39,A -85,B 0,C 180,E1 -12073.537,E2 -12073.537} C_VEL
LIN {X 0,Y 383.086,Z 501.394,A -85,B 0,C 180,E1 -12077.455,E2 -12077.455} C_VEL
LIN {X 0,Y 383.021,Z 501.396,A -85,B 0,C 180,E1 -12080.648,E2 -12080.648} C_VEL
LIN {X 0,Y 383.026,Z 501.4,A -85,B 0,C 180,E1 -12083.808,E2 -12083.808} C_VEL
LIN {X 0,Y 383.073,Z 501.391,A -85,B 0,C 180,E1 -12086.124,E2 -12086.124} C_VEL
LIN {X 0,Y 383.043,Z 501.393,A -85,B 0,C 180,E1 -12088.493,E2 -12088.493} C_VEL
LIN {X 0,Y 383.003,Z 501.399,A -85,B 0,C 180,E1 -12092.428,E2 -12092.428} C_VEL
LIN {X 0,Y 383.029,Z 501.396,A -85,B 0,C 180,E1 -12096.166,E2 -12096.166} C_VEL
LIN {X 0,Y 383.018,Z 501.399,A -85,B 0,C 180,E1 -12099.958,E2 -12099.958} C_VEL
LIN {X 0,Y 383.062,Z 501.392,A -85,B 0,C 180,E1 -12102.79,E2 -12102.79} C_VEL
LIN {X 0,Y 383.067,Z 501.395,A -85,B 0,C 180,E1 -12105.801,E2 -12105.801} C_VEL
LIN {X 0,Y 383.042,Z 501.394,A -85,B 0,C 180,E1 -12108.788,E2 -12108.788} C_VEL
LIN {X 0,Y 383.002,Z 501.4,A -85,B 0,C 180,E1 -12112.097,E2 -12112.097} C_VEL
LIN {X 0,Y 383.018,Z 501.401,A -85,B 0,C 180,E1 -12115.333,E2 -12115.333} C_VEL
LIN {X 0,Y 382.983,Z 501.403,A -85,B 0,C 180,E1 -12119.083,E2 -12119.083} C_VEL
LIN {X 0,Y 383.058,Z 501.392,A -85,B 0,C 180,E1 -12122.699,E2 -12122.699} C_VEL
LIN {X 0,Y 383.036,Z 501.396,A -85,B 0,C 180,E1 -12126.194,E2 -12126.194} C_VEL
LIN {X 0,Y 383.058,Z 501.397,A -85,B 0,C 180,E1 -12129.6,E2 -12129.6} C_VEL
LIN {X 0,Y 383.108,Z 501.386,A -85,B 0,C 180,E1 -12132.932,E2 -12132.932} C_VEL
LIN {X 0,Y 383.129,Z 501.383,A -85,B 0,C 180,E1 -12136.465,E2 -12136.465} C_VEL
LIN {X 0,Y 383.147,Z 501.381,A -85,B 0,C 180,E1 -12140.499,E2 -12140.499} C_VEL
LIN {X 0,Y 383.281,Z 501.37,A -85,B 0,C 180,E1 -12143.684,E2 -12143.684} C_VEL
LIN {X 0,Y 383.394,Z 501.354,A -85,B 0,C 180,E1 -12147.9,E2 -12147.9} C_VEL
LIN {X 0,Y 383.522,Z 501.337,A -85,B 0,C 180,E1 -12150.001,E2 -12150.001} C_VEL
LIN {X 0,Y 383.267,Z 501.368,A -85,B 0,C 180,E1 -12152.102,E2 -12152.102} C_VEL
LIN {X 0,Y 382.884,Z 501.417,A -85,B 0,C 180,E1 -12155.266,E2 -12155.266} C_VEL
LIN {X 0,Y 382.623,Z 501.512,A -85,B 0,C 180,E1 -12157.388,E2 -12157.388} C_VEL
LIN {X 0,Y 382.386,Z 504.113,A -85,B 0,C 180,E1 -12160.591,E2 -12160.591} C_VEL
LIN {X 0,Y 382.304,Z 506.387,A -85,B 0,C 180,E1 -12163.368,E2 -12163.368} C_VEL
LIN {X 0,Y 384.075,Z 511.612,A -85,B 0,C 180,E1 -12163.64,E2 -12163.64} C_VEL
LIN {X 0,Y 389.176,Z 525.75,A -85,B 0,C 180,E1 -12164.479,E2 -12164.479} C_VEL
LIN {X 0,Y 393.314,Z 539.437,A -85,B 0,C 180,E1 -12165.412,E2 -12165.412} C_VEL
LIN {X 0,Y 394.21,Z 543.471,A -85,B 0,C 180,E1 -12165.693,E2 -12165.693} C_VEL
LIN {X 0,Y 392.974,Z 558.524,A -85,B 0,C 180,E1 -12166.628,E2 -12166.628} C_VEL
LIN {X 0,Y 391.509,Z 572.968,A -85,B 0,C 180,E1 -12167.768,E2 -12167.768} C_VEL
LIN {X 0,Y 390.005,Z 586.217,A -85,B 0,C 180,E1 -12169.064,E2 -12169.064} C_VEL
LIN {X 0,Y 388.514,Z 598.441,A -85,B 0,C 180,E1 -12170.517,E2 -12170.517} C_VEL
LIN {X 0,Y 387.492,Z 605.934,A -85,B 0,C 180,E1 -12171.557,E2 -12171.557} C_VEL
LIN {X 0,Y 386.35,Z 610.107,A -85,B 0,C 180,E1 -12172.157,E2 -12172.157} C_VEL
LIN {X 0,Y 382.745,Z 616.686,A -85,B 0,C 180,E1 -12173.12,E2 -12173.12} C_VEL
LIN {X 0,Y 379.13,Z 622.895,A -85,B 0,C 180,E1 -12174.152,E2 -12174.152} C_VEL
LIN {X 0,Y 377.993,Z 626.371,A -85,B 0,C 180,E1 -12174.853,E2 -12174.853} C_VEL
LIN {X 0,Y 376.885,Z 634.834,A -85,B 0,C 180,E1 -12176.885,E2 -12176.885} C_VEL
LIN {X 0,Y 375.984,Z 642.211,A -85,B 0,C 180,E1 -12179.078,E2 -12179.078} C_VEL
LIN {X 0,Y 375.413,Z 647.526,A -85,B 0,C 180,E1 -12181.058,E2 -12181.058} C_VEL
LIN {X 0,Y 375.077,Z 651.466,A -85,B 0,C 180,E1 -12182.914,E2 -12182.914} C_VEL
LIN {X 0,Y 374.769,Z 653.918,A -85,B 0,C 180,E1 -12184.398,E2 -12184.398} C_VEL
LIN {X 0,Y 374.531,Z 656.131,A -85,B 0,C 180,E1 -12186.206,E2 -12186.206} C_VEL
LIN {X 0,Y 374.433,Z 657.661,A -85,B 0,C 180,E1 -12188.272,E2 -12188.272} C_VEL
LIN {X 0,Y 374.395,Z 658.113,A -85,B 0,C 180,E1 -12189.678,E2 -12189.678} C_VEL
LIN {X 0,Y 374.404,Z 658.062,A -85,B 0,C 180,E1 -12191.335,E2 -12191.335} C_VEL
LIN {X 0,Y 374.525,Z 657.29,A -85,B 0,C 180,E1 -12192.958,E2 -12192.958} C_VEL
LIN {X 0,Y 374.681,Z 655.955,A -85,B 0,C 180,E1 -12194.538,E2 -12194.538} C_VEL
LIN {X 0,Y 374.905,Z 654.074,A -85,B 0,C 180,E1 -12196.083,E2 -12196.083} C_VEL
LIN {X 0,Y 375.386,Z 649.839,A -85,B 0,C 180,E1 -12198.493,E2 -12198.493} C_VEL
LIN {X 0,Y 375.943,Z 644.98,A -85,B 0,C 180,E1 -12200.534,E2 -12200.534} C_VEL
LIN {X 0,Y 376.834,Z 638.526,A -85,B 0,C 180,E1 -12202.67,E2 -12202.67} C_VEL
LIN {X 0,Y 378.047,Z 630.168,A -85,B 0,C 180,E1 -12204.882,E2 -12204.882} C_VEL
LIN {X 0,Y 379.365,Z 621.288,A -85,B 0,C 180,E1 -12206.788,E2 -12206.788} C_VEL
LIN {X 0,Y 381.086,Z 610.226,A -85,B 0,C 180,E1 -12208.737,E2 -12208.737} C_VEL
LIN {X 0,Y 382.785,Z 598.483,A -85,B 0,C 180,E1 -12210.433,E2 -12210.433} C_VEL
LIN {X 0,Y 384.49,Z 585.984,A -85,B 0,C 180,E1 -12211.921,E2 -12211.921} C_VEL
LIN {X 0,Y 386.228,Z 572.142,A -85,B 0,C 180,E1 -12213.265,E2 -12213.265} C_VEL
LIN {X 0,Y 387.682,Z 559.149,A -85,B 0,C 180,E1 -12214.288,E2 -12214.288} C_VEL
LIN {X 0,Y 388.824,Z 545.678,A -85,B 0,C 180,E1 -12215.149,E2 -12215.149} C_VEL
LIN {X 0,Y 384.476,Z 531.403,A -85,B 0,C 180,E1 -12216.287,E2 -12216.287} C_VEL
LIN {X 0,Y 379.372,Z 518.513,A -85,B 0,C 180,E1 -12217.249,E2 -12217.249} C_VEL
LIN {X 0,Y 375.643,Z 510.017,A -85,B 0,C 180,E1 -12217.845,E2 -12217.845} C_VEL
LIN {X 0,Y 375.533,Z 509.334,A -85,B 0,C 180,E1 -12217.91,E2 -12217.91} C_VEL
LIN {X 0,Y 375.687,Z 506.887,A -85,B 0,C 180,E1 -12221.456,E2 -12221.456} C_VEL
LIN {X 0,Y 375.885,Z 504.648,A -85,B 0,C 180,E1 -12224.825,E2 -12224.825} C_VEL
LIN {X 0,Y 375.992,Z 503.22,A -85,B 0,C 180,E1 -12227.038,E2 -12227.038} C_VEL
LIN {X 0,Y 376.041,Z 502.274,A -85,B 0,C 180,E1 -12229.228,E2 -12229.228} C_VEL
LIN {X 0,Y 376.207,Z 502.25,A -85,B 0,C 180,E1 -12232.486,E2 -12232.486} C_VEL
LIN {X 0,Y 376.17,Z 502.254,A -85,B 0,C 180,E1 -12234.639,E2 -12234.639} C_VEL
LIN {X 0,Y 376.351,Z 502.231,A -85,B 0,C 180,E1 -12237.859,E2 -12237.859} C_VEL
LIN {X 0,Y 376.486,Z 502.214,A -85,B 0,C 180,E1 -12240,E2 -12240} C_VEL
LIN {X 0,Y 376.187,Z 502.251,A -85,B 0,C 180,E1 -12243.213,E2 -12243.213} C_VEL
LIN {X 0,Y 376.244,Z 502.244,A -85,B 0,C 180,E1 -12246.435,E2 -12246.435} C_VEL
LIN {X 0,Y 376.202,Z 502.25,A -85,B 0,C 180,E1 -12248.595,E2 -12248.595} C_VEL
LIN {X 0,Y 376.047,Z 502.267,A -85,B 0,C 180,E1 -12251.863,E2 -12251.863} C_VEL
LIN {X 0,Y 376.055,Z 502.265,A -85,B 0,C 180,E1 -12255.167,E2 -12255.167} C_VEL
LIN {X 0,Y 376.021,Z 502.274,A -85,B 0,C 180,E1 -12258.526,E2 -12258.526} C_VEL
LIN {X 0,Y 375.96,Z 502.278,A -85,B 0,C 180,E1 -12261.954,E2 -12261.954} C_VEL
LIN {X 0,Y 376.003,Z 502.273,A -85,B 0,C 180,E1 -12265.461,E2 -12265.461} C_VEL
LIN {X 0,Y 375.974,Z 502.279,A -85,B 0,C 180,E1 -12269.078,E2 -12269.078} C_VEL
LIN {X 0,Y 375.947,Z 502.282,A -85,B 0,C 180,E1 -12272.828,E2 -12272.828} C_VEL
LIN {X 0,Y 376.023,Z 502.323,A -85,B 0,C 180,E1 -12275.197,E2 -12275.197} C_VEL
LIN {X 0,Y 376.577,Z 505.548,A -85,B 0,C 180,E1 -12278.387,E2 -12278.387} C_VEL
LIN {X 0,Y 377.316,Z 509.936,A -85,B 0,C 180,E1 -12282.109,E2 -12282.109} C_VEL
LIN {X 0,Y 377.962,Z 513.801,A -85,B 0,C 180,E1 -12285.042,E2 -12285.042} C_VEL
LIN {X 0,Y 378.44,Z 517.096,A -85,B 0,C 180,E1 -12287.326,E2 -12287.326} C_VEL
LIN {X 0,Y 378.157,Z 520.802,A -85,B 0,C 180,E1 -12289.639,E2 -12289.639} C_VEL
LIN {X 0,Y 377.484,Z 527.301,A -85,B 0,C 180,E1 -12293.432,E2 -12293.432} C_VEL
LIN {X 0,Y 377,Z 531.971,A -85,B 0,C 180,E1 -12295.996,E2 -12295.996} C_VEL
LIN {X 0,Y 376.476,Z 538.019,A -85,B 0,C 180,E1 -12299.173,E2 -12299.173} C_VEL
LIN {X 0,Y 376.022,Z 543.91,A -85,B 0,C 180,E1 -12302.143,E2 -12302.143} C_VEL
LIN {X 0,Y 376.929,Z 547.292,A -85,B 0,C 180,E1 -12302.315,E2 -12302.315} C_VEL
LIN {X 0,Y 381.237,Z 562.244,A -85,B 0,C 180,E1 -12303.151,E2 -12303.151} C_VEL
LIN {X 0,Y 384.283,Z 576.7,A -85,B 0,C 180,E1 -12304.049,E2 -12304.049} C_VEL
LIN {X 0,Y 386.215,Z 590.544,A -85,B 0,C 180,E1 -12305.013,E2 -12305.013} C_VEL
LIN {X 0,Y 386.655,Z 595.512,A -85,B 0,C 180,E1 -12305.385,E2 -12305.385} C_VEL
LIN {X 0,Y 385.169,Z 608.768,A -85,B 0,C 180,E1 -12306.333,E2 -12306.333} C_VEL
LIN {X 0,Y 383.485,Z 622.1,A -85,B 0,C 180,E1 -12307.507,E2 -12307.507} C_VEL
LIN {X 0,Y 381.643,Z 635.521,A -85,B 0,C 180,E1 -12308.955,E2 -12308.955} C_VEL
LIN {X 0,Y 380.228,Z 645.833,A -85,B 0,C 180,E1 -12310.286,E2 -12310.286} C_VEL
LIN {X 0,Y 378.804,Z 656.381,A -85,B 0,C 180,E1 -12311.894,E2 -12311.894} C_VEL
LIN {X 0,Y 377.557,Z 665.368,A -85,B 0,C 180,E1 -12313.508,E2 -12313.508} C_VEL
LIN {X 0,Y 376.477,Z 674.266,A -85,B 0,C 180,E1 -12315.403,E2 -12315.403} C_VEL
LIN {X 0,Y 375.582,Z 682.655,A -85,B 0,C 180,E1 -12317.573,E2 -12317.573} C_VEL
LIN {X 0,Y 374.97,Z 689.397,A -85,B 0,C 180,E1 -12319.743,E2 -12319.743} C_VEL
LIN {X 0,Y 374.728,Z 694.695,A -85,B 0,C 180,E1 -12321.913,E2 -12321.913} C_VEL
LIN {X 0,Y 374.591,Z 698.434,A -85,B 0,C 180,E1 -12323.918,E2 -12323.918} C_VEL
LIN {X 0,Y 374.569,Z 700.775,A -85,B 0,C 180,E1 -12325.695,E2 -12325.695} C_VEL
LIN {X 0,Y 374.674,Z 702.571,A -85,B 0,C 180,E1 -12327.85,E2 -12327.85} C_VEL
LIN {X 0,Y 374.663,Z 703.187,A -85,B 0,C 180,E1 -12329.999,E2 -12329.999} C_VEL
LIN {X 0,Y 374.673,Z 702.595,A -85,B 0,C 180,E1 -12332.149,E2 -12332.149} C_VEL
LIN {X 0,Y 374.568,Z 700.782,A -85,B 0,C 180,E1 -12334.304,E2 -12334.304} C_VEL
LIN {X 0,Y 374.673,Z 697.766,A -85,B 0,C 180,E1 -12336.461,E2 -12336.461} C_VEL
LIN {X 0,Y 374.784,Z 693.462,A -85,B 0,C 180,E1 -12338.627,E2 -12338.627} C_VEL
LIN {X 0,Y 375.106,Z 687.765,A -85,B 0,C 180,E1 -12340.798,E2 -12340.798} C_VEL
LIN {X 0,Y 375.726,Z 680.53,A -85,B 0,C 180,E1 -12342.97,E2 -12342.97} C_VEL
LIN {X 0,Y 376.749,Z 671.548,A -85,B 0,C 180,E1 -12345.138,E2 -12345.138} C_VEL
LIN {X 0,Y 377.87,Z 661.982,A -85,B 0,C 180,E1 -12347.033,E2 -12347.033} C_VEL
LIN {X 0,Y 379.32,Z 651.241,A -85,B 0,C 180,E1 -12348.796,E2 -12348.796} C_VEL
LIN {X 0,Y 380.786,Z 639.636,A -85,B 0,C 180,E1 -12350.387,E2 -12350.387} C_VEL
LIN {X 0,Y 382.52,Z 626.749,A -85,B 0,C 180,E1 -12351.841,E2 -12351.841} C_VEL
LIN {X 0,Y 384.023,Z 614.032,A -85,B 0,C 180,E1 -12353.027,E2 -12353.027} C_VEL
LIN {X 0,Y 385.565,Z 600.687,A -85,B 0,C 180,E1 -12354.038,E2 -12354.038} C_VEL
LIN {X 0,Y 386.085,Z 594.074,A -85,B 0,C 180,E1 -12354.473,E2 -12354.473} C_VEL
LIN {X 0,Y 384.015,Z 580.398,A -85,B 0,C 180,E1 -12355.413,E2 -12355.413} C_VEL
LIN {X 0,Y 380.754,Z 564.736,A -85,B 0,C 180,E1 -12356.329,E2 -12356.329} C_VEL
LIN {X 0,Y 376.598,Z 548.94,A -85,B 0,C 180,E1 -12357.089,E2 -12357.089} C_VEL
LIN {X 0,Y 376.043,Z 546.291,A -85,B 0,C 180,E1 -12357.195,E2 -12357.195} C_VEL
LIN {X 0,Y 376.631,Z 538.95,A -85,B 0,C 180,E1 -12360.867,E2 -12360.867} C_VEL
LIN {X 0,Y 377.169,Z 532.918,A -85,B 0,C 180,E1 -12363.986,E2 -12363.986} C_VEL
LIN {X 0,Y 377.818,Z 525.641,A -85,B 0,C 180,E1 -12367.867,E2 -12367.867} C_VEL
LIN {X 0,Y 378.352,Z 520.812,A -85,B 0,C 180,E1 -12370.55,E2 -12370.55} C_VEL
LIN {X 0,Y 378.519,Z 517.19,A -85,B 0,C 180,E1 -12372.662,E2 -12372.662} C_VEL
LIN {X 0,Y 377.986,Z 513.338,A -85,B 0,C 180,E1 -12375.046,E2 -12375.046} C_VEL
LIN {X 0,Y 377.08,Z 508.558,A -85,B 0,C 180,E1 -12378.202,E2 -12378.202} C_VEL
LIN {X 0,Y 376.146,Z 503.269,A -85,B 0,C 180,E1 -12381.934,E2 -12381.934} C_VEL
LIN {X 0,Y 375.954,Z 502.281,A -85,B 0,C 180,E1 -12382.756,E2 -12382.756} C_VEL
LIN {X 0,Y 375.951,Z 502.28,A -85,B 0,C 180,E1 -12385.888,E2 -12385.888} C_VEL
LIN {X 0,Y 375.959,Z 502.28,A -85,B 0,C 180,E1 -12389.687,E2 -12389.687} C_VEL
LIN {X 0,Y 375.993,Z 502.272,A -85,B 0,C 180,E1 -12392.141,E2 -12392.141} C_VEL
LIN {X 0,Y 375.996,Z 502.271,A -85,B 0,C 180,E1 -12394.539,E2 -12394.539} C_VEL
LIN {X 0,Y 375.948,Z 502.279,A -85,B 0,C 180,E1 -12398.045,E2 -12398.045} C_VEL
LIN {X 0,Y 376.014,Z 502.275,A -85,B 0,C 180,E1 -12401.474,E2 -12401.474} C_VEL
LIN {X 0,Y 376.052,Z 502.265,A -85,B 0,C 180,E1 -12404.833,E2 -12404.833} C_VEL
LIN {X 0,Y 376.049,Z 502.266,A -85,B 0,C 180,E1 -12408.137,E2 -12408.137} C_VEL
LIN {X 0,Y 376.248,Z 502.243,A -85,B 0,C 180,E1 -12411.878,E2 -12411.878} C_VEL
LIN {X 0,Y 376.165,Z 502.25,A -85,B 0,C 180,E1 -12414.64,E2 -12414.64} C_VEL
LIN {X 0,Y 376.345,Z 502.231,A -85,B 0,C 180,E1 -12417.86,E2 -12417.86} C_VEL
LIN {X 0,Y 376.481,Z 502.213,A -85,B 0,C 180,E1 -12420,E2 -12420} C_VEL
LIN {X 0,Y 376.185,Z 502.251,A -85,B 0,C 180,E1 -12423.213,E2 -12423.213} C_VEL
LIN {X 0,Y 376.229,Z 502.242,A -85,B 0,C 180,E1 -12426.557,E2 -12426.557} C_VEL
LIN {X 0,Y 376.11,Z 502.262,A -85,B 0,C 180,E1 -12429.682,E2 -12429.682} C_VEL
LIN {X 0,Y 376.081,Z 502.266,A -85,B 0,C 180,E1 -12433.658,E2 -12433.658} C_VEL
LIN {X 0,Y 376.035,Z 502.272,A -85,B 0,C 180,E1 -12437.608,E2 -12437.608} C_VEL
LIN {X 0,Y 375.97,Z 502.275,A -85,B 0,C 180,E1 -12440.833,E2 -12440.833} C_VEL
LIN {X 0,Y 375.986,Z 502.273,A -85,B 0,C 180,E1 -12444.283,E2 -12444.283} C_VEL
LIN {X 0,Y 376.013,Z 502.269,A -85,B 0,C 180,E1 -12446.653,E2 -12446.653} C_VEL
LIN {X 0,Y 375.971,Z 502.276,A -85,B 0,C 180,E1 -12449.08,E2 -12449.08} C_VEL
LIN {X 0,Y 375.951,Z 502.277,A -85,B 0,C 180,E1 -12452.829,E2 -12452.829} C_VEL
LIN {X 0,Y 375.953,Z 502.282,A -85,B 0,C 180,E1 -12455.417,E2 -12455.417} C_VEL
LIN {X 0,Y 375.974,Z 502.274,A -85,B 0,C 180,E1 -12458.273,E2 -12458.273} C_VEL
LIN {X 0,Y 375.986,Z 502.278,A -85,B 0,C 180,E1 -12461.612,E2 -12461.612} C_VEL
LIN {X 0,Y 376.012,Z 502.272,A -85,B 0,C 180,E1 -12465.256,E2 -12465.256} C_VEL
LIN {X 0,Y 375.987,Z 502.272,A -85,B 0,C 180,E1 -12468.391,E2 -12468.391} C_VEL
LIN {X 0,Y 375.967,Z 502.278,A -85,B 0,C 180,E1 -12471.913,E2 -12471.913} C_VEL
LIN {X 0,Y 375.979,Z 502.277,A -85,B 0,C 180,E1 -12475.334,E2 -12475.334} C_VEL
LIN {X 0,Y 375.958,Z 502.276,A -85,B 0,C 180,E1 -12478.439,E2 -12478.439} C_VEL
LIN {X 0,Y 375.997,Z 502.272,A -85,B 0,C 180,E1 -12482.143,E2 -12482.143} C_VEL
LIN {X 0,Y 376.008,Z 502.27,A -85,B 0,C 180,E1 -12484.54,E2 -12484.54} C_VEL
LIN {X 0,Y 375.966,Z 502.277,A -85,B 0,C 180,E1 -12488.047,E2 -12488.047} C_VEL
LIN {X 0,Y 376.027,Z 502.273,A -85,B 0,C 180,E1 -12491.475,E2 -12491.475} C_VEL
LIN {X 0,Y 376.062,Z 502.263,A -85,B 0,C 180,E1 -12494.834,E2 -12494.834} C_VEL
LIN {X 0,Y 376.053,Z 502.266,A -85,B 0,C 180,E1 -12498.137,E2 -12498.137} C_VEL
LIN {X 0,Y 376.205,Z 502.248,A -85,B 0,C 180,E1 -12501.939,E2 -12501.939} C_VEL
LIN {X 0,Y 376.174,Z 502.249,A -85,B 0,C 180,E1 -12504.641,E2 -12504.641} C_VEL
LIN {X 0,Y 376.36,Z 502.23,A -85,B 0,C 180,E1 -12507.86,E2 -12507.86} C_VEL
LIN {X 0,Y 376.491,Z 502.212,A -85,B 0,C 180,E1 -12510.001,E2 -12510.001} C_VEL
LIN {X 0,Y 376.205,Z 502.247,A -85,B 0,C 180,E1 -12512.142,E2 -12512.142} C_VEL
LIN {X 0,Y 375.831,Z 502.296,A -85,B 0,C 180,E1 -12515.365,E2 -12515.365} C_VEL
LIN {X 0,Y 375.554,Z 502.477,A -85,B 0,C 180,E1 -12517.528,E2 -12517.528} C_VEL
LIN {X 0,Y 375.317,Z 505.1,A -85,B 0,C 180,E1 -12520.793,E2 -12520.793} C_VEL
LIN {X 0,Y 375.314,Z 506.784,A -85,B 0,C 180,E1 -12522.874,E2 -12522.874} C_VEL
LIN {X 0,Y 376.942,Z 511.755,A -85,B 0,C 180,E1 -12523.135,E2 -12523.135} C_VEL
LIN {X 0,Y 382.489,Z 526.992,A -85,B 0,C 180,E1 -12524.069,E2 -12524.069} C_VEL
LIN {X 0,Y 386.632,Z 540.773,A -85,B 0,C 180,E1 -12525.04,E2 -12525.04} C_VEL
LIN {X 0,Y 387.601,Z 545.102,A -85,B 0,C 180,E1 -12525.358,E2 -12525.358} C_VEL
LIN {X 0,Y 386.399,Z 558.975,A -85,B 0,C 180,E1 -12526.239,E2 -12526.239} C_VEL
LIN {X 0,Y 384.912,Z 573.316,A -85,B 0,C 180,E1 -12527.391,E2 -12527.391} C_VEL
LIN {X 0,Y 383.325,Z 586.645,A -85,B 0,C 180,E1 -12528.715,E2 -12528.715} C_VEL
LIN {X 0,Y 381.806,Z 598.577,A -85,B 0,C 180,E1 -12530.152,E2 -12530.152} C_VEL
LIN {X 0,Y 380.324,Z 609.282,A -85,B 0,C 180,E1 -12531.69,E2 -12531.69} C_VEL
LIN {X 0,Y 378.918,Z 619.761,A -85,B 0,C 180,E1 -12533.502,E2 -12533.502} C_VEL
LIN {X 0,Y 377.993,Z 626.371,A -85,B 0,C 180,E1 -12534.853,E2 -12534.853} C_VEL
LIN {X 0,Y 376.89,Z 629.734,A -85,B 0,C 180,E1 -12535.575,E2 -12535.575} C_VEL
LIN {X 0,Y 373.423,Z 634.952,A -85,B 0,C 180,E1 -12536.748,E2 -12536.748} C_VEL
LIN {X 0,Y 370.022,Z 639.733,A -85,B 0,C 180,E1 -12537.983,E2 -12537.983} C_VEL
LIN {X 0,Y 369.04,Z 642.319,A -85,B 0,C 180,E1 -12538.793,E2 -12538.793} C_VEL
LIN {X 0,Y 368.355,Z 648.155,A -85,B 0,C 180,E1 -12541.007,E2 -12541.007} C_VEL
LIN {X 0,Y 368.025,Z 651.94,A -85,B 0,C 180,E1 -12542.833,E2 -12542.833} C_VEL
LIN {X 0,Y 367.585,Z 655.257,A -85,B 0,C 180,E1 -12545,E2 -12545} C_VEL
LIN {X 0,Y 367.428,Z 656.95,A -85,B 0,C 180,E1 -12546.547,E2 -12546.547} C_VEL
LIN {X 0,Y 367.341,Z 658.121,A -85,B 0,C 180,E1 -12548.332,E2 -12548.332} C_VEL
LIN {X 0,Y 367.305,Z 658.583,A -85,B 0,C 180,E1 -12550.583,E2 -12550.583} C_VEL
LIN {X 0,Y 367.362,Z 658.243,A -85,B 0,C 180,E1 -12552.035,E2 -12552.035} C_VEL
LIN {X 0,Y 367.479,Z 657.403,A -85,B 0,C 180,E1 -12553.511,E2 -12553.511} C_VEL
LIN {X 0,Y 367.77,Z 655.081,A -85,B 0,C 180,E1 -12555.775,E2 -12555.775} C_VEL
LIN {X 0,Y 368.241,Z 651.383,A -85,B 0,C 180,E1 -12558.101,E2 -12558.101} C_VEL
LIN {X 0,Y 368.841,Z 646.372,A -85,B 0,C 180,E1 -12560.386,E2 -12560.386} C_VEL
LIN {X 0,Y 369.733,Z 640.267,A -85,B 0,C 180,E1 -12562.535,E2 -12562.535} C_VEL
LIN {X 0,Y 370.805,Z 633.024,A -85,B 0,C 180,E1 -12564.586,E2 -12564.586} C_VEL
LIN {X 0,Y 372.107,Z 624.69,A -85,B 0,C 180,E1 -12566.522,E2 -12566.522} C_VEL
LIN {X 0,Y 373.686,Z 615.001,A -85,B 0,C 180,E1 -12568.382,E2 -12568.382} C_VEL
LIN {X 0,Y 375.402,Z 604.213,A -85,B 0,C 180,E1 -12570.102,E2 -12570.102} C_VEL
LIN {X 0,Y 377.152,Z 592.7,A -85,B 0,C 180,E1 -12571.629,E2 -12571.629} C_VEL
LIN {X 0,Y 378.774,Z 580.792,A -85,B 0,C 180,E1 -12572.95,E2 -12572.95} C_VEL
LIN {X 0,Y 380.487,Z 567.024,A -85,B 0,C 180,E1 -12574.195,E2 -12574.195} C_VEL
LIN {X 0,Y 381.976,Z 553.585,A -85,B 0,C 180,E1 -12575.169,E2 -12575.169} C_VEL
LIN {X 0,Y 382.446,Z 548.221,A -85,B 0,C 180,E1 -12575.498,E2 -12575.498} C_VEL
LIN {X 0,Y 379.129,Z 536.349,A -85,B 0,C 180,E1 -12576.486,E2 -12576.486} C_VEL
LIN {X 0,Y 374.103,Z 522.801,A -85,B 0,C 180,E1 -12577.567,E2 -12577.567} C_VEL
LIN {X 0,Y 368.71,Z 510.858,A -85,B 0,C 180,E1 -12578.47,E2 -12578.47} C_VEL
LIN {X 0,Y 368.533,Z 509.864,A -85,B 0,C 180,E1 -12578.558,E2 -12578.558} C_VEL
LIN {X 0,Y 368.716,Z 507.297,A -85,B 0,C 180,E1 -12582.369,E2 -12582.369} C_VEL
LIN {X 0,Y 368.961,Z 504.798,A -85,B 0,C 180,E1 -12586.274,E2 -12586.274} C_VEL
LIN {X 0,Y 368.97,Z 503.155,A -85,B 0,C 180,E1 -12589.019,E2 -12589.019} C_VEL
LIN {X 0,Y 369.161,Z 503.128,A -85,B 0,C 180,E1 -12592.341,E2 -12592.341} C_VEL
LIN {X 0,Y 369.142,Z 503.13,A -85,B 0,C 180,E1 -12594.537,E2 -12594.537} C_VEL
LIN {X 0,Y 369.316,Z 503.107,A -85,B 0,C 180,E1 -12597.818,E2 -12597.818} C_VEL
LIN {X 0,Y 369.455,Z 503.089,A -85,B 0,C 180,E1 -12600,E2 -12600} C_VEL
LIN {X 0,Y 369.316,Z 503.107,A -85,B 0,C 180,E1 -12602.181,E2 -12602.181} C_VEL
LIN {X 0,Y 369.206,Z 503.121,A -85,B 0,C 180,E1 -12606.558,E2 -12606.558} C_VEL
LIN {X 0,Y 369.135,Z 503.13,A -85,B 0,C 180,E1 -12608.761,E2 -12608.761} C_VEL
LIN {X 0,Y 369.003,Z 503.145,A -85,B 0,C 180,E1 -12612.093,E2 -12612.093} C_VEL
LIN {X 0,Y 368.994,Z 503.144,A -85,B 0,C 180,E1 -12615.465,E2 -12615.465} C_VEL
LIN {X 0,Y 368.964,Z 503.149,A -85,B 0,C 180,E1 -12618.893,E2 -12618.893} C_VEL
LIN {X 0,Y 368.929,Z 503.157,A -85,B 0,C 180,E1 -12622.395,E2 -12622.395} C_VEL
LIN {X 0,Y 368.997,Z 503.149,A -85,B 0,C 180,E1 -12625.98,E2 -12625.98} C_VEL
LIN {X 0,Y 368.965,Z 503.151,A -85,B 0,C 180,E1 -12628.813,E2 -12628.813} C_VEL
LIN {X 0,Y 368.897,Z 503.161,A -85,B 0,C 180,E1 -12632.238,E2 -12632.238} C_VEL
LIN {X 0,Y 368.894,Z 503.16,A -85,B 0,C 180,E1 -12633.538,E2 -12633.538} C_VEL
LIN {X 0,Y 369.05,Z 503.738,A -85,B 0,C 180,E1 -12635.029,E2 -12635.029} C_VEL
LIN {X 0,Y 369.716,Z 507.568,A -85,B 0,C 180,E1 -12638.851,E2 -12638.851} C_VEL
LIN {X 0,Y 370.394,Z 511.551,A -85,B 0,C 180,E1 -12642.269,E2 -12642.269} C_VEL
LIN {X 0,Y 371.204,Z 516.491,A -85,B 0,C 180,E1 -12646.009,E2 -12646.009} C_VEL
LIN {X 0,Y 371.441,Z 518.751,A -85,B 0,C 180,E1 -12647.554,E2 -12647.554} C_VEL
LIN {X 0,Y 371.093,Z 522.457,A -85,B 0,C 180,E1 -12649.916,E2 -12649.916} C_VEL
LIN {X 0,Y 370.485,Z 528.321,A -85,B 0,C 180,E1 -12653.394,E2 -12653.394} C_VEL
LIN {X 0,Y 369.825,Z 534.32,A -85,B 0,C 180,E1 -12656.736,E2 -12656.736} C_VEL
LIN {X 0,Y 369.338,Z 539.922,A -85,B 0,C 180,E1 -12659.718,E2 -12659.718} C_VEL
LIN {X 0,Y 369.048,Z 543.387,A -85,B 0,C 180,E1 -12661.503,E2 -12661.503} C_VEL
LIN {X 0,Y 370.01,Z 546.856,A -85,B 0,C 180,E1 -12661.687,E2 -12661.687} C_VEL
LIN {X 0,Y 374.414,Z 561.769,A -85,B 0,C 180,E1 -12662.568,E2 -12662.568} C_VEL
LIN {X 0,Y 377.86,Z 577.999,A -85,B 0,C 180,E1 -12663.625,E2 -12663.625} C_VEL
LIN {X 0,Y 379.717,Z 592.05,A -85,B 0,C 180,E1 -12664.646,E2 -12664.646} C_VEL
LIN {X 0,Y 380.12,Z 595.831,A -85,B 0,C 180,E1 -12664.952,E2 -12664.952} C_VEL
LIN {X 0,Y 378.443,Z 610.265,A -85,B 0,C 180,E1 -12666.031,E2 -12666.031} C_VEL
LIN {X 0,Y 376.532,Z 624.502,A -85,B 0,C 180,E1 -12667.358,E2 -12667.358} C_VEL
LIN {X 0,Y 374.812,Z 636.343,A -85,B 0,C 180,E1 -12668.697,E2 -12668.697} C_VEL
LIN {X 0,Y 373.205,Z 647.422,A -85,B 0,C 180,E1 -12670.186,E2 -12670.186} C_VEL
LIN {X 0,Y 371.76,Z 657.706,A -85,B 0,C 180,E1 -12671.824,E2 -12671.824} C_VEL
LIN {X 0,Y 370.314,Z 667.786,A -85,B 0,C 180,E1 -12673.744,E2 -12673.744} C_VEL
LIN {X 0,Y 369.256,Z 676.213,A -85,B 0,C 180,E1 -12675.674,E2 -12675.674} C_VEL
LIN {X 0,Y 368.396,Z 684.146,A -85,B 0,C 180,E1 -12677.886,E2 -12677.886} C_VEL
LIN {X 0,Y 367.813,Z 690.483,A -85,B 0,C 180,E1 -12680.097,E2 -12680.097} C_VEL
LIN {X 0,Y 367.603,Z 695.409,A -85,B 0,C 180,E1 -12682.309,E2 -12682.309} C_VEL
LIN {X 0,Y 367.48,Z 699.022,A -85,B 0,C 180,E1 -12684.512,E2 -12684.512} C_VEL
LIN {X 0,Y 367.458,Z 701.399,A -85,B 0,C 180,E1 -12686.71,E2 -12686.71} C_VEL
LIN {X 0,Y 367.598,Z 702.599,A -85,B 0,C 180,E1 -12688.904,E2 -12688.904} C_VEL
LIN {X 0,Y 367.598,Z 702.616,A -85,B 0,C 180,E1 -12691.095,E2 -12691.095} C_VEL
LIN {X 0,Y 367.588,Z 702.158,A -85,B 0,C 180,E1 -12692.191,E2 -12692.191} C_VEL
LIN {X 0,Y 367.497,Z 700.331,A -85,B 0,C 180,E1 -12694.387,E2 -12694.387} C_VEL
LIN {X 0,Y 367.575,Z 697.298,A -85,B 0,C 180,E1 -12696.587,E2 -12696.587} C_VEL
LIN {X 0,Y 367.717,Z 692.977,A -85,B 0,C 180,E1 -12698.794,E2 -12698.794} C_VEL
LIN {X 0,Y 368.08,Z 687.261,A -85,B 0,C 180,E1 -12701.007,E2 -12701.007} C_VEL
LIN {X 0,Y 368.695,Z 680.001,A -85,B 0,C 180,E1 -12703.222,E2 -12703.222} C_VEL
LIN {X 0,Y 369.666,Z 672.247,A -85,B 0,C 180,E1 -12705.153,E2 -12705.153} C_VEL
LIN {X 0,Y 370.799,Z 662.909,A -85,B 0,C 180,E1 -12707.084,E2 -12707.084} C_VEL
LIN {X 0,Y 372.29,Z 652.248,A -85,B 0,C 180,E1 -12708.908,E2 -12708.908} C_VEL
LIN {X 0,Y 373.785,Z 641.144,A -85,B 0,C 180,E1 -12710.498,E2 -12710.498} C_VEL
LIN {X 0,Y 375.369,Z 629.888,A -85,B 0,C 180,E1 -12711.845,E2 -12711.845} C_VEL
LIN {X 0,Y 377.032,Z 616.399,A -85,B 0,C 180,E1 -12713.189,E2 -12713.189} C_VEL
LIN {X 0,Y 378.821,Z 601.933,A -85,B 0,C 180,E1 -12714.339,E2 -12714.339} C_VEL
LIN {X 0,Y 379.383,Z 595.065,A -85,B 0,C 180,E1 -12714.809,E2 -12714.809} C_VEL
LIN {X 0,Y 377.132,Z 580.302,A -85,B 0,C 180,E1 -12715.856,E2 -12715.856} C_VEL
LIN {X 0,Y 373.932,Z 564.925,A -85,B 0,C 180,E1 -12716.78,E2 -12716.78} C_VEL
LIN {X 0,Y 369.666,Z 548.611,A -85,B 0,C 180,E1 -12717.594,E2 -12717.594} C_VEL
LIN {X 0,Y 369.072,Z 545.896,A -85,B 0,C 180,E1 -12717.725,E2 -12717.725} C_VEL
LIN {X 0,Y 369.623,Z 539.158,A -85,B 0,C 180,E1 -12721.171,E2 -12721.171} C_VEL
LIN {X 0,Y 370.224,Z 532.451,A -85,B 0,C 180,E1 -12724.713,E2 -12724.713} C_VEL
LIN {X 0,Y 371.092,Z 524.557,A -85,B 0,C 180,E1 -12729.061,E2 -12729.061} C_VEL
LIN {X 0,Y 371.499,Z 520.395,A -85,B 0,C 180,E1 -12731.461,E2 -12731.461} C_VEL
LIN {X 0,Y 371.492,Z 517.958,A -85,B 0,C 180,E1 -12732.925,E2 -12732.925} C_VEL
LIN {X 0,Y 370.889,Z 513.946,A -85,B 0,C 180,E1 -12735.484,E2 -12735.484} C_VEL
LIN {X 0,Y 369.801,Z 508.081,A -85,B 0,C 180,E1 -12739.479,E2 -12739.479} C_VEL
LIN {X 0,Y 368.929,Z 503.168,A -85,B 0,C 180,E1 -12743.091,E2 -12743.091} C_VEL
LIN {X 0,Y 368.888,Z 503.159,A -85,B 0,C 180,E1 -12746.461,E2 -12746.461} C_VEL
LIN {X 0,Y 368.914,Z 503.153,A -85,B 0,C 180,E1 -12750.31,E2 -12750.31} C_VEL
LIN {X 0,Y 368.973,Z 503.152,A -85,B 0,C 180,E1 -12753.535,E2 -12753.535} C_VEL
LIN {X 0,Y 368.947,Z 503.149,A -85,B 0,C 180,E1 -12756.421,E2 -12756.421} C_VEL
LIN {X 0,Y 368.927,Z 503.154,A -85,B 0,C 180,E1 -12759.947,E2 -12759.947} C_VEL
LIN {X 0,Y 368.969,Z 503.152,A -85,B 0,C 180,E1 -12763.399,E2 -12763.399} C_VEL
LIN {X 0,Y 369.05,Z 503.137,A -85,B 0,C 180,E1 -12766.79,E2 -12766.79} C_VEL
LIN {X 0,Y 369.062,Z 503.136,A -85,B 0,C 180,E1 -12770.132,E2 -12770.132} C_VEL
LIN {X 0,Y 369.178,Z 503.12,A -85,B 0,C 180,E1 -12772.343,E2 -12772.343} C_VEL
LIN {X 0,Y 369.138,Z 503.125,A -85,B 0,C 180,E1 -12774.538,E2 -12774.538} C_VEL
LIN {X 0,Y 369.31,Z 503.107,A -85,B 0,C 180,E1 -12777.819,E2 -12777.819} C_VEL
LIN {X 0,Y 369.45,Z 503.088,A -85,B 0,C 180,E1 -12780,E2 -12780} C_VEL
LIN {X 0,Y 369.311,Z 503.105,A -85,B 0,C 180,E1 -12782.182,E2 -12782.182} C_VEL
LIN {X 0,Y 369.199,Z 503.118,A -85,B 0,C 180,E1 -12786.559,E2 -12786.559} C_VEL
LIN {X 0,Y 369.059,Z 503.138,A -85,B 0,C 180,E1 -12789.869,E2 -12789.869} C_VEL
LIN {X 0,Y 369.028,Z 503.143,A -85,B 0,C 180,E1 -12793.773,E2 -12793.773} C_VEL
LIN {X 0,Y 368.993,Z 503.148,A -85,B 0,C 180,E1 -12797.769,E2 -12797.769} C_VEL
LIN {X 0,Y 368.921,Z 503.155,A -85,B 0,C 180,E1 -12801.221,E2 -12801.221} C_VEL
LIN {X 0,Y 368.951,Z 503.149,A -85,B 0,C 180,E1 -12804.776,E2 -12804.776} C_VEL
LIN {X 0,Y 368.98,Z 503.145,A -85,B 0,C 180,E1 -12808.437,E2 -12808.437} C_VEL
LIN {X 0,Y 368.904,Z 503.155,A -85,B 0,C 180,E1 -12812.238,E2 -12812.238} C_VEL
LIN {X 0,Y 368.924,Z 503.153,A -85,B 0,C 180,E1 -12815.003,E2 -12815.003} C_VEL
LIN {X 0,Y 368.909,Z 503.154,A -85,B 0,C 180,E1 -12818.643,E2 -12818.643} C_VEL
LIN {X 0,Y 368.938,Z 503.152,A -85,B 0,C 180,E1 -12822.021,E2 -12822.021} C_VEL
LIN {X 0,Y 368.987,Z 503.147,A -85,B 0,C 180,E1 -12825.194,E2 -12825.194} C_VEL
LIN {X 0,Y 368.943,Z 503.15,A -85,B 0,C 180,E1 -12828.188,E2 -12828.188} C_VEL
LIN {X 0,Y 368.912,Z 503.157,A -85,B 0,C 180,E1 -12831.36,E2 -12831.36} C_VEL
LIN {X 0,Y 368.936,Z 503.153,A -85,B 0,C 180,E1 -12835.148,E2 -12835.148} C_VEL
LIN {X 0,Y 368.929,Z 503.153,A -85,B 0,C 180,E1 -12839.048,E2 -12839.048} C_VEL
LIN {X 0,Y 368.981,Z 503.151,A -85,B 0,C 180,E1 -12841.565,E2 -12841.565} C_VEL
LIN {X 0,Y 369.001,Z 503.145,A -85,B 0,C 180,E1 -12844.021,E2 -12844.021} C_VEL
LIN {X 0,Y 368.935,Z 503.157,A -85,B 0,C 180,E1 -12847.606,E2 -12847.606} C_VEL
LIN {X 0,Y 368.985,Z 503.146,A -85,B 0,C 180,E1 -12851.108,E2 -12851.108} C_VEL
LIN {X 0,Y 369.002,Z 503.142,A -85,B 0,C 180,E1 -12854.536,E2 -12854.536} C_VEL
LIN {X 0,Y 369.009,Z 503.145,A -85,B 0,C 180,E1 -12857.908,E2 -12857.908} C_VEL
LIN {X 0,Y 369.152,Z 503.127,A -85,B 0,C 180,E1 -12861.89,E2 -12861.89} C_VEL
LIN {X 0,Y 369.146,Z 503.124,A -85,B 0,C 180,E1 -12864.538,E2 -12864.538} C_VEL
LIN {X 0,Y 369.324,Z 503.107,A -85,B 0,C 180,E1 -12867.819,E2 -12867.819} C_VEL
LIN {X 0,Y 369.46,Z 503.088,A -85,B 0,C 180,E1 -12870.001,E2 -12870.001} C_VEL
LIN {X 0,Y 369.146,Z 503.126,A -85,B 0,C 180,E1 -12872.183,E2 -12872.183} C_VEL
LIN {X 0,Y 368.763,Z 503.177,A -85,B 0,C 180,E1 -12875.469,E2 -12875.469} C_VEL
LIN {X 0,Y 368.479,Z 503.445,A -85,B 0,C 180,E1 -12877.673,E2 -12877.673} C_VEL
LIN {X 0,Y 368.253,Z 506.108,A -85,B 0,C 180,E1 -12881.003,E2 -12881.003} C_VEL
LIN {X 0,Y 368.264,Z 507.182,A -85,B 0,C 180,E1 -12882.355,E2 -12882.355} C_VEL
LIN {X 0,Y 369.279,Z 510.305,A -85,B 0,C 180,E1 -12882.524,E2 -12882.524} C_VEL
LIN {X 0,Y 374.954,Z 525.784,A -85,B 0,C 180,E1 -12883.481,E2 -12883.481} C_VEL
LIN {X 0,Y 379.082,Z 538.935,A -85,B 0,C 180,E1 -12884.417,E2 -12884.417} C_VEL
LIN {X 0,Y 381.011,Z 545.947,A -85,B 0,C 180,E1 -12884.966,E2 -12884.966} C_VEL
LIN {X 0,Y 379.72,Z 560.34,A -85,B 0,C 180,E1 -12885.909,E2 -12885.909} C_VEL
LIN {X 0,Y 378.301,Z 573.787,A -85,B 0,C 180,E1 -12887.014,E2 -12887.014} C_VEL
LIN {X 0,Y 376.863,Z 585.55,A -85,B 0,C 180,E1 -12888.183,E2 -12888.183} C_VEL
LIN {X 0,Y 375.221,Z 598.176,A -85,B 0,C 180,E1 -12889.703,E2 -12889.703} C_VEL
LIN {X 0,Y 373.667,Z 608.727,A -85,B 0,C 180,E1 -12891.227,E2 -12891.227} C_VEL
LIN {X 0,Y 372.138,Z 619.632,A -85,B 0,C 180,E1 -12893.117,E2 -12893.117} C_VEL
LIN {X 0,Y 370.679,Z 629.696,A -85,B 0,C 180,E1 -12895.252,E2 -12895.252} C_VEL
LIN {X 0,Y 369.592,Z 638.086,A -85,B 0,C 180,E1 -12897.46,E2 -12897.46} C_VEL
LIN {X 0,Y 369.04,Z 642.319,A -85,B 0,C 180,E1 -12898.793,E2 -12898.793} C_VEL
LIN {X 0,Y 368.099,Z 644.766,A -85,B 0,C 180,E1 -12899.617,E2 -12899.617} C_VEL
LIN {X 0,Y 363.487,Z 649.837,A -85,B 0,C 180,E1 -12901.51,E2 -12901.51} C_VEL
LIN {X 0,Y 361.29,Z 652.232,A -85,B 0,C 180,E1 -12902.655,E2 -12902.655} C_VEL
LIN {X 0,Y 360.827,Z 653.239,A -85,B 0,C 180,E1 -12903.257,E2 -12903.257} C_VEL
LIN {X 0,Y 360.507,Z 655.818,A -85,B 0,C 180,E1 -12905.036,E2 -12905.036} C_VEL
LIN {X 0,Y 360.308,Z 657.892,A -85,B 0,C 180,E1 -12907.205,E2 -12907.205} C_VEL
LIN {X 0,Y 360.258,Z 658.723,A -85,B 0,C 180,E1 -12908.708,E2 -12908.708} C_VEL
LIN {X 0,Y 360.215,Z 659.032,A -85,B 0,C 180,E1 -12910.454,E2 -12910.454} C_VEL
LIN {X 0,Y 360.284,Z 658.654,A -85,B 0,C 180,E1 -12912.16,E2 -12912.16} C_VEL
LIN {X 0,Y 360.509,Z 657.018,A -85,B 0,C 180,E1 -12914.572,E2 -12914.572} C_VEL
LIN {X 0,Y 360.928,Z 653.95,A -85,B 0,C 180,E1 -12917.037,E2 -12917.037} C_VEL
LIN {X 0,Y 361.458,Z 649.803,A -85,B 0,C 180,E1 -12919.314,E2 -12919.314} C_VEL
LIN {X 0,Y 362.264,Z 644.194,A -85,B 0,C 180,E1 -12921.624,E2 -12921.624} C_VEL
LIN {X 0,Y 363.264,Z 637.669,A -85,B 0,C 180,E1 -12923.743,E2 -12923.743} C_VEL
LIN {X 0,Y 364.493,Z 630.421,A -85,B 0,C 180,E1 -12925.668,E2 -12925.668} C_VEL
LIN {X 0,Y 366.023,Z 621.37,A -85,B 0,C 180,E1 -12927.655,E2 -12927.655} C_VEL
LIN {X 0,Y 367.717,Z 611.377,A -85,B 0,C 180,E1 -12929.471,E2 -12929.471} C_VEL
LIN {X 0,Y 369.573,Z 600.018,A -85,B 0,C 180,E1 -12931.181,E2 -12931.181} C_VEL
LIN {X 0,Y 371.502,Z 587.243,A -85,B 0,C 180,E1 -12932.764,E2 -12932.764} C_VEL
LIN {X 0,Y 373.249,Z 574.756,A -85,B 0,C 180,E1 -12934.037,E2 -12934.037} C_VEL
LIN {X 0,Y 374.964,Z 560.611,A -85,B 0,C 180,E1 -12935.204,E2 -12935.204} C_VEL
LIN {X 0,Y 376.065,Z 549.566,A -85,B 0,C 180,E1 -12935.944,E2 -12935.944} C_VEL
LIN {X 0,Y 372.045,Z 535.923,A -85,B 0,C 180,E1 -12937.143,E2 -12937.143} C_VEL
LIN {X 0,Y 366.726,Z 522.326,A -85,B 0,C 180,E1 -12938.277,E2 -12938.277} C_VEL
LIN {X 0,Y 361.693,Z 511.273,A -85,B 0,C 180,E1 -12939.16,E2 -12939.16} C_VEL
LIN {X 0,Y 361.547,Z 510.412,A -85,B 0,C 180,E1 -12939.236,E2 -12939.236} C_VEL
LIN {X 0,Y 361.716,Z 507.921,A -85,B 0,C 180,E1 -12943.055,E2 -12943.055} C_VEL
LIN {X 0,Y 361.967,Z 505.754,A -85,B 0,C 180,E1 -12946.526,E2 -12946.526} C_VEL
LIN {X 0,Y 361.955,Z 504.416,A -85,B 0,C 180,E1 -12948.803,E2 -12948.803} C_VEL
LIN {X 0,Y 362.051,Z 504.013,A -85,B 0,C 180,E1 -12951.066,E2 -12951.066} C_VEL
LIN {X 0,Y 362.161,Z 503.999,A -85,B 0,C 180,E1 -12953.313,E2 -12953.313} C_VEL
LIN {X 0,Y 362.281,Z 503.984,A -85,B 0,C 180,E1 -12957.776,E2 -12957.776} C_VEL
LIN {X 0,Y 362.425,Z 503.965,A -85,B 0,C 180,E1 -12960,E2 -12960} C_VEL
LIN {X 0,Y 362.28,Z 503.984,A -85,B 0,C 180,E1 -12962.223,E2 -12962.223} C_VEL
LIN {X 0,Y 362.17,Z 503.998,A -85,B 0,C 180,E1 -12966.686,E2 -12966.686} C_VEL
LIN {X 0,Y 362.071,Z 504.008,A -85,B 0,C 180,E1 -12968.933,E2 -12968.933} C_VEL
LIN {X 0,Y 361.958,Z 504.023,A -85,B 0,C 180,E1 -12972.332,E2 -12972.332} C_VEL
LIN {X 0,Y 361.959,Z 504.024,A -85,B 0,C 180,E1 -12974.62,E2 -12974.62} C_VEL
LIN {X 0,Y 361.954,Z 504.023,A -85,B 0,C 180,E1 -12978.099,E2 -12978.099} C_VEL
LIN {X 0,Y 361.889,Z 504.03,A -85,B 0,C 180,E1 -12981.653,E2 -12981.653} C_VEL
LIN {X 0,Y 361.925,Z 504.026,A -85,B 0,C 180,E1 -12985.29,E2 -12985.29} C_VEL
LIN {X 0,Y 361.92,Z 504.031,A -85,B 0,C 180,E1 -12987.778,E2 -12987.778} C_VEL
LIN {X 0,Y 361.844,Z 504.039,A -85,B 0,C 180,E1 -12991.285,E2 -12991.285} C_VEL
LIN {X 0,Y 361.856,Z 504.036,A -85,B 0,C 180,E1 -12993.369,E2 -12993.369} C_VEL
LIN {X 0,Y 362.215,Z 505.824,A -85,B 0,C 180,E1 -12995.597,E2 -12995.597} C_VEL
LIN {X 0,Y 362.838,Z 509.469,A -85,B 0,C 180,E1 -12999.215,E2 -12999.215} C_VEL
LIN {X 0,Y 363.512,Z 513.523,A -85,B 0,C 180,E1 -13002.72,E2 -13002.72} C_VEL
LIN {X 0,Y 364.245,Z 517.825,A -85,B 0,C 180,E1 -13006.004,E2 -13006.004} C_VEL
LIN {X 0,Y 364.449,Z 520.003,A -85,B 0,C 180,E1 -13007.551,E2 -13007.551} C_VEL
LIN {X 0,Y 363.957,Z 524.706,A -85,B 0,C 180,E1 -13010.569,E2 -13010.569} C_VEL
LIN {X 0,Y 363.272,Z 531.342,A -85,B 0,C 180,E1 -13014.522,E2 -13014.522} C_VEL
LIN {X 0,Y 362.507,Z 538.57,A -85,B 0,C 180,E1 -13018.543,E2 -13018.543} C_VEL
LIN {X 0,Y 362.079,Z 542.86,A -85,B 0,C 180,E1 -13020.83,E2 -13020.83} C_VEL
LIN {X 0,Y 363.089,Z 546.416,A -85,B 0,C 180,E1 -13021.028,E2 -13021.028} C_VEL
LIN {X 0,Y 367.516,Z 560.876,A -85,B 0,C 180,E1 -13021.93,E2 -13021.93} C_VEL
LIN {X 0,Y 370.862,Z 576.106,A -85,B 0,C 180,E1 -13022.957,E2 -13022.957} C_VEL
LIN {X 0,Y 372.88,Z 590.083,A -85,B 0,C 180,E1 -13024.003,E2 -13024.003} C_VEL
LIN {X 0,Y 373.56,Z 596.957,A -85,B 0,C 180,E1 -13024.561,E2 -13024.561} C_VEL
LIN {X 0,Y 371.961,Z 610.22,A -85,B 0,C 180,E1 -13025.587,E2 -13025.587} C_VEL
LIN {X 0,Y 370.149,Z 623.088,A -85,B 0,C 180,E1 -13026.798,E2 -13026.798} C_VEL
LIN {X 0,Y 368.159,Z 636.155,A -85,B 0,C 180,E1 -13028.293,E2 -13028.293} C_VEL
LIN {X 0,Y 366.46,Z 647.165,A -85,B 0,C 180,E1 -13029.805,E2 -13029.805} C_VEL
LIN {X 0,Y 364.931,Z 657.394,A -85,B 0,C 180,E1 -13031.472,E2 -13031.472} C_VEL
LIN {X 0,Y 363.402,Z 667.45,A -85,B 0,C 180,E1 -13033.426,E2 -13033.426} C_VEL
LIN {X 0,Y 362.312,Z 675.871,A -85,B 0,C 180,E1 -13035.394,E2 -13035.394} C_VEL
LIN {X 0,Y 361.364,Z 683.784,A -85,B 0,C 180,E1 -13037.647,E2 -13037.647} C_VEL
LIN {X 0,Y 360.747,Z 690.107,A -85,B 0,C 180,E1 -13039.901,E2 -13039.901} C_VEL
LIN {X 0,Y 360.515,Z 695.014,A -85,B 0,C 180,E1 -13042.156,E2 -13042.156} C_VEL
LIN {X 0,Y 360.398,Z 698.614,A -85,B 0,C 180,E1 -13044.404,E2 -13044.404} C_VEL
LIN {X 0,Y 360.373,Z 700.983,A -85,B 0,C 180,E1 -13046.645,E2 -13046.645} C_VEL
LIN {X 0,Y 360.533,Z 702.173,A -85,B 0,C 180,E1 -13048.882,E2 -13048.882} C_VEL
LIN {X 0,Y 360.532,Z 702.182,A -85,B 0,C 180,E1 -13051.116,E2 -13051.116} C_VEL
LIN {X 0,Y 360.371,Z 700.945,A -85,B 0,C 180,E1 -13053.353,E2 -13053.353} C_VEL
LIN {X 0,Y 360.437,Z 698.512,A -85,B 0,C 180,E1 -13055.594,E2 -13055.594} C_VEL
LIN {X 0,Y 360.557,Z 694.829,A -85,B 0,C 180,E1 -13057.841,E2 -13057.841} C_VEL
LIN {X 0,Y 360.749,Z 689.803,A -85,B 0,C 180,E1 -13060.097,E2 -13060.097} C_VEL
LIN {X 0,Y 361.342,Z 683.321,A -85,B 0,C 180,E1 -13062.353,E2 -13062.353} C_VEL
LIN {X 0,Y 362.24,Z 675.198,A -85,B 0,C 180,E1 -13064.608,E2 -13064.608} C_VEL
LIN {X 0,Y 363.341,Z 666.542,A -85,B 0,C 180,E1 -13066.576,E2 -13066.576} C_VEL
LIN {X 0,Y 364.661,Z 657.779,A -85,B 0,C 180,E1 -13068.25,E2 -13068.25} C_VEL
LIN {X 0,Y 366.196,Z 646.616,A -85,B 0,C 180,E1 -13070.038,E2 -13070.038} C_VEL
LIN {X 0,Y 367.8,Z 635.067,A -85,B 0,C 180,E1 -13071.581,E2 -13071.581} C_VEL
LIN {X 0,Y 369.507,Z 622.722,A -85,B 0,C 180,E1 -13072.948,E2 -13072.948} C_VEL
LIN {X 0,Y 371.284,Z 609.313,A -85,B 0,C 180,E1 -13074.162,E2 -13074.162} C_VEL
LIN {X 0,Y 372.653,Z 596.039,A -85,B 0,C 180,E1 -13075.144,E2 -13075.144} C_VEL
LIN {X 0,Y 370.481,Z 581.483,A -85,B 0,C 180,E1 -13076.219,E2 -13076.219} C_VEL
LIN {X 0,Y 367.568,Z 567.101,A -85,B 0,C 180,E1 -13077.13,E2 -13077.13} C_VEL
LIN {X 0,Y 363.531,Z 551.239,A -85,B 0,C 180,E1 -13077.978,E2 -13077.978} C_VEL
LIN {X 0,Y 362.07,Z 545.444,A -85,B 0,C 180,E1 -13078.276,E2 -13078.276} C_VEL
LIN {X 0,Y 362.726,Z 537.997,A -85,B 0,C 180,E1 -13082.195,E2 -13082.195} C_VEL
LIN {X 0,Y 363.346,Z 531.657,A -85,B 0,C 180,E1 -13085.671,E2 -13085.671} C_VEL
LIN {X 0,Y 364.138,Z 524.768,A -85,B 0,C 180,E1 -13089.56,E2 -13089.56} C_VEL
LIN {X 0,Y 364.446,Z 521.923,A -85,B 0,C 180,E1 -13091.23,E2 -13091.23} C_VEL
LIN {X 0,Y 364.502,Z 519.202,A -85,B 0,C 180,E1 -13092.889,E2 -13092.889} C_VEL
LIN {X 0,Y 363.88,Z 515.014,A -85,B 0,C 180,E1 -13095.61,E2 -13095.61} C_VEL
LIN {X 0,Y 362.935,Z 510.04,A -85,B 0,C 180,E1 -13099.042,E2 -13099.042} C_VEL
LIN {X 0,Y 362.062,Z 505.07,A -85,B 0,C 180,E1 -13102.734,E2 -13102.734} C_VEL
LIN {X 0,Y 361.868,Z 504.035,A -85,B 0,C 180,E1 -13103.676,E2 -13103.676} C_VEL
LIN {X 0,Y 361.84,Z 504.037,A -85,B 0,C 180,E1 -13107.055,E2 -13107.055} C_VEL
LIN {X 0,Y 361.893,Z 504.029,A -85,B 0,C 180,E1 -13110.955,E2 -13110.955} C_VEL
LIN {X 0,Y 361.946,Z 504.027,A -85,B 0,C 180,E1 -13113.475,E2 -13113.475} C_VEL
LIN {X 0,Y 361.873,Z 504.033,A -85,B 0,C 180,E1 -13117.144,E2 -13117.144} C_VEL
LIN {X 0,Y 361.911,Z 504.026,A -85,B 0,C 180,E1 -13120.724,E2 -13120.724} C_VEL
LIN {X 0,Y 361.939,Z 504.022,A -85,B 0,C 180,E1 -13124.226,E2 -13124.226} C_VEL
LIN {X 0,Y 361.99,Z 504.015,A -85,B 0,C 180,E1 -13126.528,E2 -13126.528} C_VEL
LIN {X 0,Y 362.026,Z 504.013,A -85,B 0,C 180,E1 -13129.938,E2 -13129.938} C_VEL
LIN {X 0,Y 362.141,Z 503.997,A -85,B 0,C 180,E1 -13132.193,E2 -13132.193} C_VEL
LIN {X 0,Y 362.111,Z 504,A -85,B 0,C 180,E1 -13134.432,E2 -13134.432} C_VEL
LIN {X 0,Y 362.274,Z 503.984,A -85,B 0,C 180,E1 -13137.777,E2 -13137.777} C_VEL
LIN {X 0,Y 362.42,Z 503.964,A -85,B 0,C 180,E1 -13140,E2 -13140} C_VEL
LIN {X 0,Y 362.275,Z 503.981,A -85,B 0,C 180,E1 -13142.224,E2 -13142.224} C_VEL
